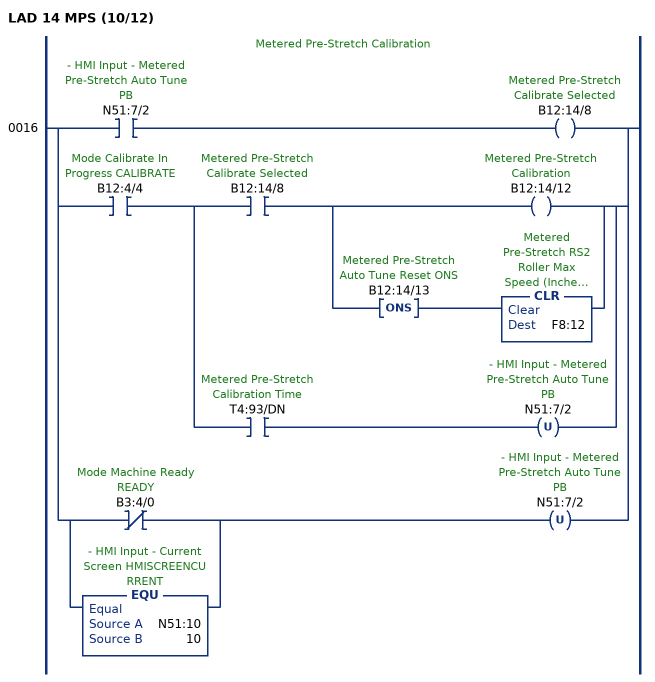
% Rung: 16 %
% Metered Pre-Stretch Calibration %
SOR BST XIC N51:7/2 OTE B12:14/8 NXB XIC B12:4/4 BST XIC B12:14/8 BST OTE B12:14/12 NXB ONS B12:14/13 CLR F8:12 BND NXB XIC T4:93/DN OTU N51:7/2 BND NXB BST XIO B3:4/0 NXB EQU N51:10 10 BND OTU N51:7/2 BND EOR
%   N51:7/2  "- HMI Input - Metered Pre-Stretch Auto Tune PB" %
%   B12:14/8  "Metered Pre-Stretch Calibrate Selected" %
%   B12:4/4  CALIBRATE  "Mode Calibrate In Progress" %
%   B12:14/12  "Metered Pre-Stretch Calibration" %
%   B12:14/13  "Metered Pre-Stretch Auto Tune Reset ONS" %
%   F8:12  RS2MAXSPEED  "Metered Pre-Stretch RS2 Roller Max Speed (Inches Per Second)" %
%   T4:93  "Metered Pre-Stretch Calibration Time" %
%   B3:4/0  READY  "Mode Machine Ready" %
%   N51:10  HMISCREENCURRENT  "- HMI Input - Current Screen" %

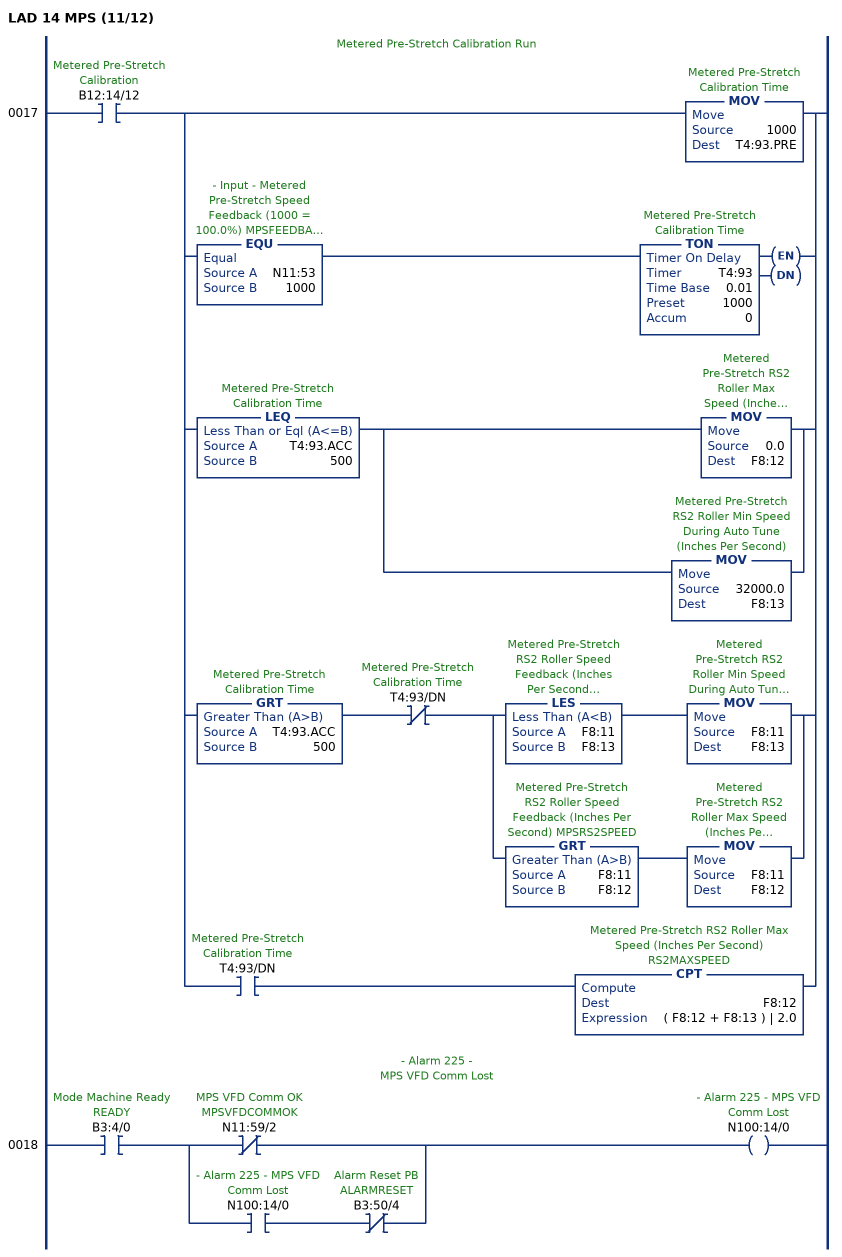
% Rung: 17 %
% Metered Pre-Stretch Calibration Run %
SOR XIC B12:14/12 BST MOV 1000 T4:93.PRE NXB EQU N11:53 1000 TON T4:93 0.01 1000 0 NXB LEQ T4:93.ACC 500 BST MOV 0.0 F8:12 NXB MOV 32000.0 F8:13 BND NXB GRT T4:93.ACC 500 XIO T4:93/DN BST LES F8:11 F8:13 MOV F8:11 F8:13 NXB GRT F8:11 F8:12 MOV F8:11 F8:12 BND NXB XIC T4:93/DN CPT F8:12 " ( F8:12 + F8:13 ) | 2.0 " BND EOR
%   B12:14/12  "Metered Pre-Stretch Calibration" %
%   T4:93  "Metered Pre-Stretch Calibration Time" %
%   N11:53  MPSFEEDBACK  "- Input - Metered Pre-Stretch Speed Feedback (1000 = 100.0%)" %
%   F8:12  RS2MAXSPEED  "Metered Pre-Stretch RS2 Roller Max Speed (Inches Per Second)" %
%   F8:13  "Metered Pre-Stretch RS2 Roller Min Speed During Auto Tune (Inches Per Second)" %
%   F8:11  MPSRS2SPEED  "Metered Pre-Stretch RS2 Roller Speed Feedback (Inches Per Second)" %
% Rung: 18 %
% - Alarm 225 -
% 
% MPS VFD Comm Lost %
SOR XIC B3:4/0 BST XIO N11:59/2 NXB XIC N100:14/0 XIO B3:50/4 BND OTE N100:14/0 EOR
%   B3:4/0  READY  "Mode Machine Ready" %
%   N11:59/2  MPSVFDCOMMOK  "MPS VFD Comm OK" %
%   N100:14/0  "- Alarm 225 - MPS VFD Comm Lost" %
%   B3:50/4  ALARMRESET  "Alarm Reset PB" %

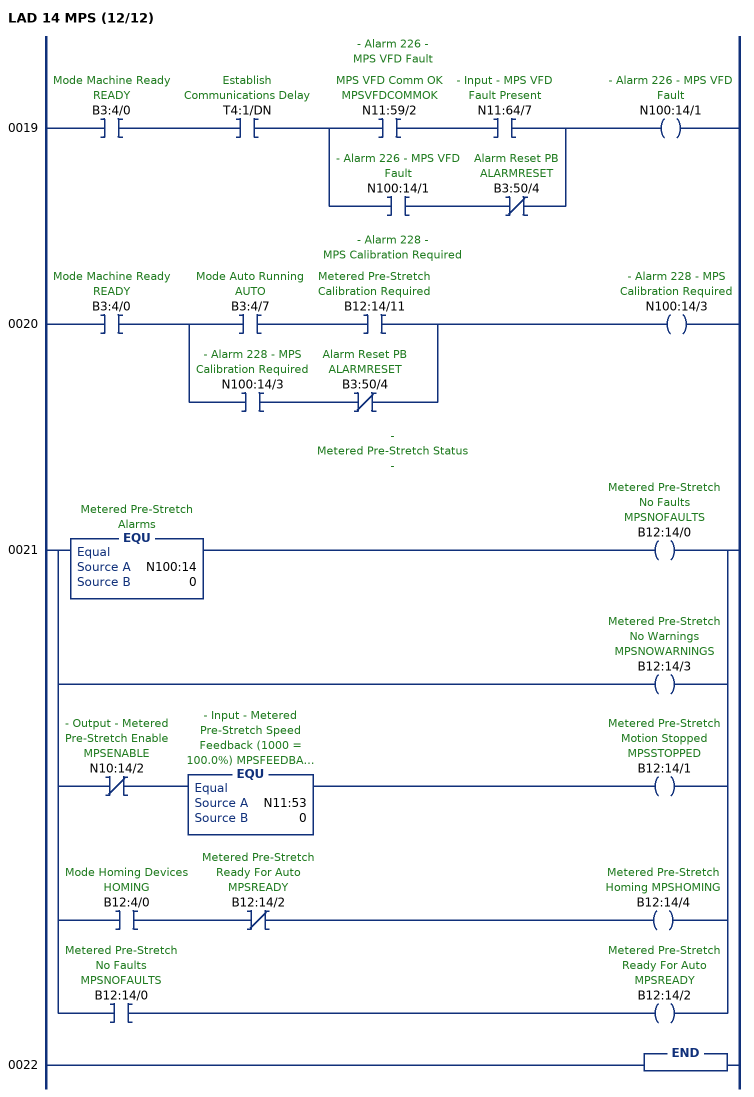
% Rung: 19 %
% - Alarm 226 -
% 
% MPS VFD Fault %
SOR XIC B3:4/0 XIC T4:1/DN BST XIC N11:59/2 XIC N11:64/7 NXB XIC N100:14/1 XIO B3:50/4 BND OTE N100:14/1 EOR
%   B3:4/0  READY  "Mode Machine Ready" %
%   T4:1  "Establish Communications Delay" %
%   N11:59/2  MPSVFDCOMMOK  "MPS VFD Comm OK" %
%   N11:64/7  "- Input - MPS VFD Fault Present" %
%   N100:14/1  "- Alarm 226 - MPS VFD Fault" %
%   B3:50/4  ALARMRESET  "Alarm Reset PB" %
% Rung: 20 %
% - Alarm 228 -
% 
% MPS Calibration Required %
SOR XIC B3:4/0 BST XIC B3:4/7 XIC B12:14/11 NXB XIC N100:14/3 XIO B3:50/4 BND OTE N100:14/3 EOR
%   B3:4/0  READY  "Mode Machine Ready" %
%   B3:4/7  AUTO  "Mode Auto Running" %
%   B12:14/11  "Metered Pre-Stretch Calibration Required" %
%   N100:14/3  "- Alarm 228 - MPS Calibration Required" %
%   B3:50/4  ALARMRESET  "Alarm Reset PB" %
% Rung: 21 %
% -
% 
% Metered Pre-Stretch Status
% 
% - %
SOR BST EQU N100:14 0 OTE B12:14/0 NXB OTE B12:14/3 NXB XIO N10:14/2 EQU N11:53 0 OTE B12:14/1 NXB XIC B12:4/0 XIO B12:14/2 OTE B12:14/4 NXB XIC B12:14/0 OTE B12:14/2 BND EOR
%   N100:14  "Metered Pre-Stretch Alarms" %
%   B12:14/0  MPSNOFAULTS  "Metered Pre-Stretch No Faults" %
%   B12:14/3  MPSNOWARNINGS  "Metered Pre-Stretch No Warnings" %
%   N10:14/2  MPSENABLE  "- Output - Metered Pre-Stretch Enable" %
%   N11:53  MPSFEEDBACK  "- Input - Metered Pre-Stretch Speed Feedback (1000 = 100.0%)" %
%   B12:14/1  MPSSTOPPED  "Metered Pre-Stretch Motion Stopped" %
%   B12:4/0  HOMING  "Mode Homing Devices" %
%   B12:14/2  MPSREADY  "Metered Pre-Stretch Ready For Auto" %
%   B12:14/4  MPSHOMING  "Metered Pre-Stretch Homing" %
% Rung: 22 %
SOR END EOR

LADDER 15 "CUTTER ASM"
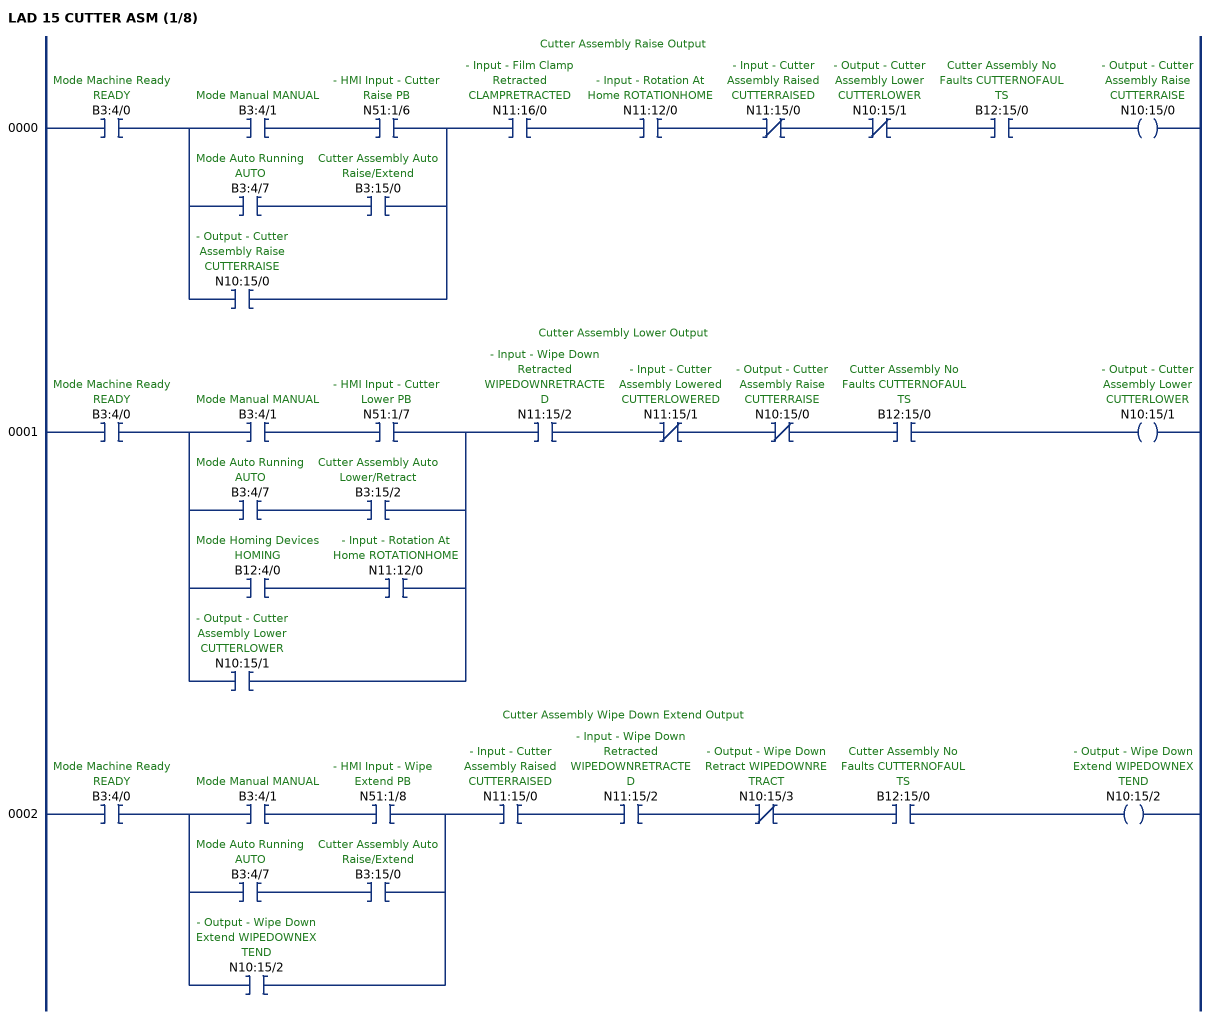
% Rung: 0 %
% Cutter Assembly Raise Output %
SOR XIC B3:4/0 BST XIC B3:4/1 XIC N51:1/6 NXB XIC B3:4/7 XIC B3:15/0 NXB XIC N10:15/0 BND XIC N11:16/0 XIC N11:12/0 XIO N11:15/0 XIO N10:15/1 XIC B12:15/0 OTE N10:15/0 EOR
%   B3:4/0  READY  "Mode Machine Ready" %
%   B3:4/1  MANUAL  "Mode Manual" %
%   N51:1/6  "- HMI Input - Cutter Raise PB" %
%   B3:4/7  AUTO  "Mode Auto Running" %
%   B3:15/0  "Cutter Assembly Auto Raise/Extend" %
%   N10:15/0  CUTTERRAISE  "- Output - Cutter Assembly Raise" %
%   N11:16/0  CLAMPRETRACTED  "- Input - Film Clamp Retracted" %
%   N11:12/0  ROTATIONHOME  "- Input - Rotation At Home" %
%   N11:15/0  CUTTERRAISED  "- Input - Cutter Assembly Raised" %
%   N10:15/1  CUTTERLOWER  "- Output - Cutter Assembly Lower" %
%   B12:15/0  CUTTERNOFAULTS  "Cutter Assembly No Faults" %
% Rung: 1 %
% Cutter Assembly Lower Output %
SOR XIC B3:4/0 BST XIC B3:4/1 XIC N51:1/7 NXB XIC B3:4/7 XIC B3:15/2 NXB XIC B12:4/0 XIC N11:12/0 NXB XIC N10:15/1 BND XIC N11:15/2 XIO N11:15/1 XIO N10:15/0 XIC B12:15/0 OTE N10:15/1 EOR
%   B3:4/0  READY  "Mode Machine Ready" %
%   B3:4/1  MANUAL  "Mode Manual" %
%   N51:1/7  "- HMI Input - Cutter Lower PB" %
%   B3:4/7  AUTO  "Mode Auto Running" %
%   B3:15/2  "Cutter Assembly Auto Lower/Retract" %
%   B12:4/0  HOMING  "Mode Homing Devices" %
%   N11:12/0  ROTATIONHOME  "- Input - Rotation At Home" %
%   N10:15/1  CUTTERLOWER  "- Output - Cutter Assembly Lower" %
%   N11:15/2  WIPEDOWNRETRACTED  "- Input - Wipe Down Retracted" %
%   N11:15/1  CUTTERLOWERED  "- Input - Cutter Assembly Lowered" %
%   N10:15/0  CUTTERRAISE  "- Output - Cutter Assembly Raise" %
%   B12:15/0  CUTTERNOFAULTS  "Cutter Assembly No Faults" %
% Rung: 2 %
% Cutter Assembly Wipe Down Extend Output %
SOR XIC B3:4/0 BST XIC B3:4/1 XIC N51:1/8 NXB XIC B3:4/7 XIC B3:15/0 NXB XIC N10:15/2 BND XIC N11:15/0 XIC N11:15/2 XIO N10:15/3 XIC B12:15/0 OTE N10:15/2 EOR
%   B3:4/0  READY  "Mode Machine Ready" %
%   B3:4/1  MANUAL  "Mode Manual" %
%   N51:1/8  "- HMI Input - Wipe Extend PB" %
%   B3:4/7  AUTO  "Mode Auto Running" %
%   B3:15/0  "Cutter Assembly Auto Raise/Extend" %
%   N10:15/2  WIPEDOWNEXTEND  "- Output - Wipe Down Extend" %
%   N11:15/0  CUTTERRAISED  "- Input - Cutter Assembly Raised" %
%   N11:15/2  WIPEDOWNRETRACTED  "- Input - Wipe Down Retracted" %
%   N10:15/3  WIPEDOWNRETRACT  "- Output - Wipe Down Retract" %
%   B12:15/0  CUTTERNOFAULTS  "Cutter Assembly No Faults" %

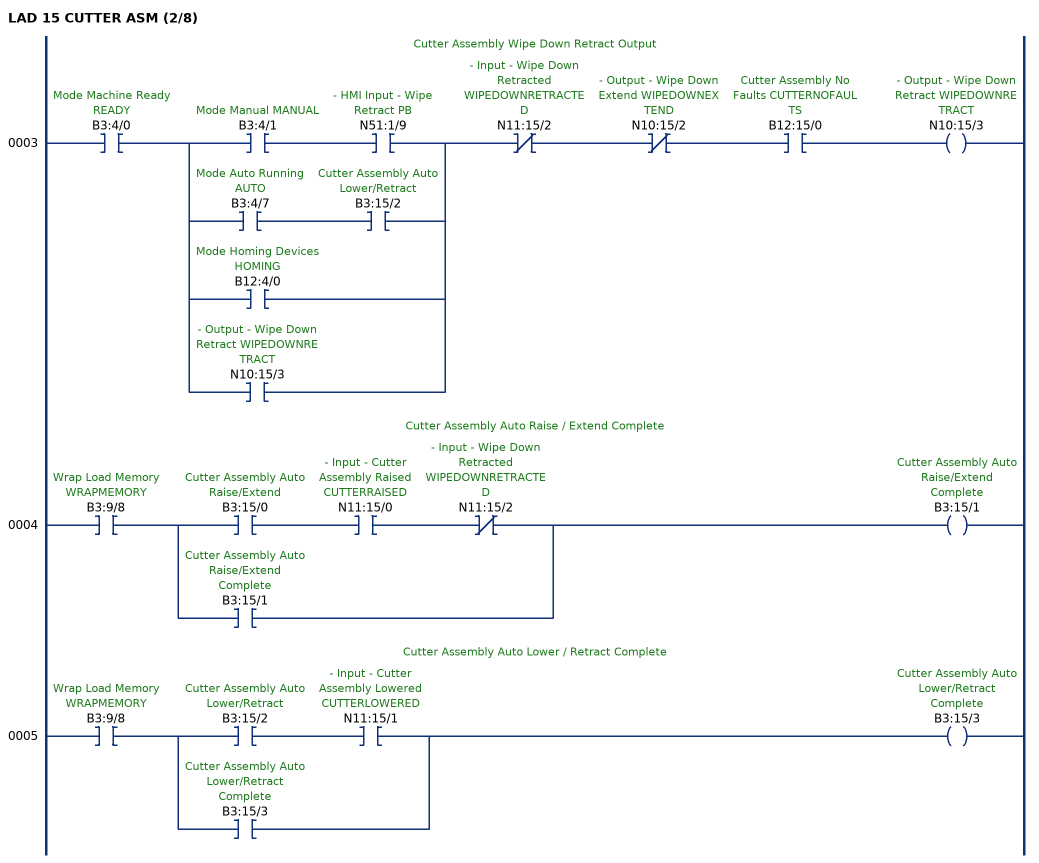
% Rung: 3 %
% Cutter Assembly Wipe Down Retract Output %
SOR XIC B3:4/0 BST XIC B3:4/1 XIC N51:1/9 NXB XIC B3:4/7 XIC B3:15/2 NXB XIC B12:4/0 NXB XIC N10:15/3 BND XIO N11:15/2 XIO N10:15/2 XIC B12:15/0 OTE N10:15/3 EOR
%   B3:4/0  READY  "Mode Machine Ready" %
%   B3:4/1  MANUAL  "Mode Manual" %
%   N51:1/9  "- HMI Input - Wipe Retract PB" %
%   B3:4/7  AUTO  "Mode Auto Running" %
%   B3:15/2  "Cutter Assembly Auto Lower/Retract" %
%   B12:4/0  HOMING  "Mode Homing Devices" %
%   N10:15/3  WIPEDOWNRETRACT  "- Output - Wipe Down Retract" %
%   N11:15/2  WIPEDOWNRETRACTED  "- Input - Wipe Down Retracted" %
%   N10:15/2  WIPEDOWNEXTEND  "- Output - Wipe Down Extend" %
%   B12:15/0  CUTTERNOFAULTS  "Cutter Assembly No Faults" %
% Rung: 4 %
% Cutter Assembly Auto Raise / Extend Complete %
SOR XIC B3:9/8 BST XIC B3:15/0 XIC N11:15/0 XIO N11:15/2 NXB XIC B3:15/1 BND OTE B3:15/1 EOR
%   B3:9/8  WRAPMEMORY  "Wrap Load Memory" %
%   B3:15/0  "Cutter Assembly Auto Raise/Extend" %
%   N11:15/0  CUTTERRAISED  "- Input - Cutter Assembly Raised" %
%   N11:15/2  WIPEDOWNRETRACTED  "- Input - Wipe Down Retracted" %
%   B3:15/1  "Cutter Assembly Auto Raise/Extend Complete" %
% Rung: 5 %
% Cutter Assembly Auto Lower / Retract Complete %
SOR XIC B3:9/8 BST XIC B3:15/2 XIC N11:15/1 NXB XIC B3:15/3 BND OTE B3:15/3 EOR
%   B3:9/8  WRAPMEMORY  "Wrap Load Memory" %
%   B3:15/2  "Cutter Assembly Auto Lower/Retract" %
%   N11:15/1  CUTTERLOWERED  "- Input - Cutter Assembly Lowered" %
%   B3:15/3  "Cutter Assembly Auto Lower/Retract Complete" %

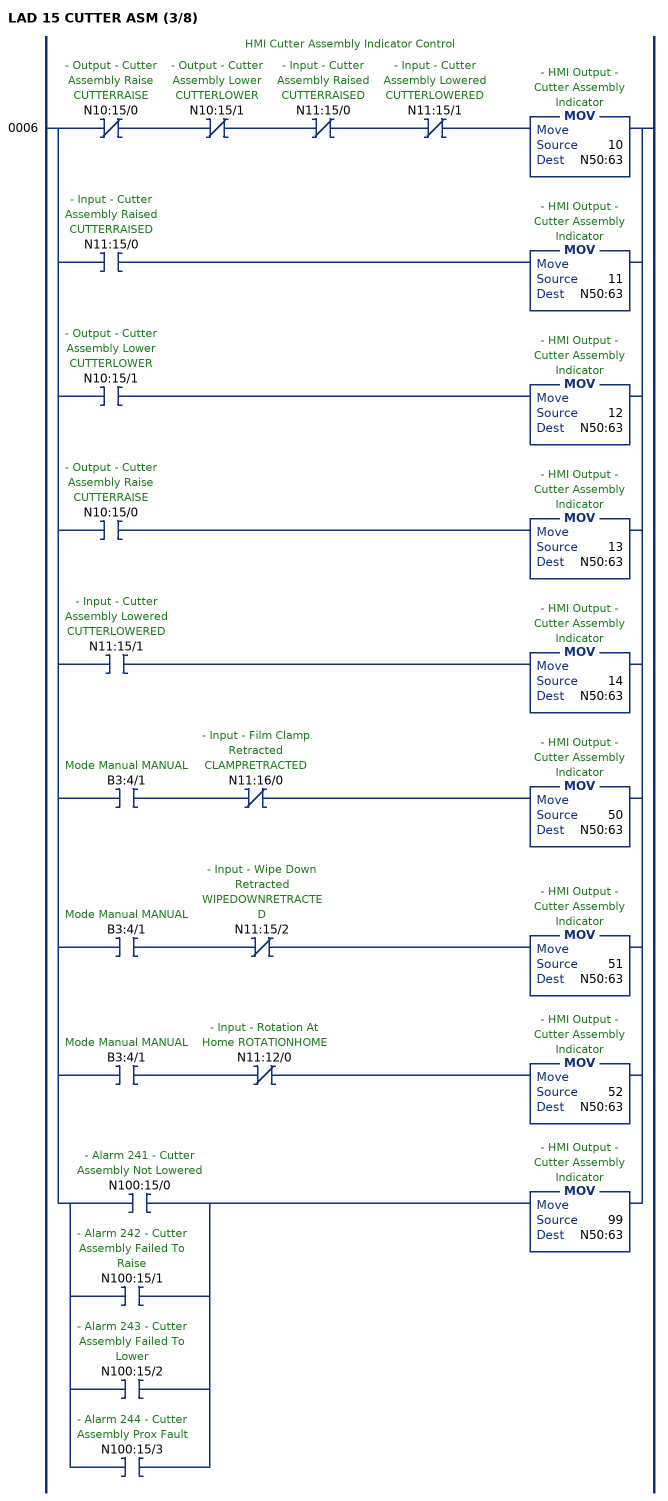
% Rung: 6 %
% HMI Cutter Assembly Indicator Control %
SOR BST XIO N10:15/0 XIO N10:15/1 XIO N11:15/0 XIO N11:15/1 MOV 10 N50:63 NXB XIC N11:15/0 MOV 11 N50:63 NXB XIC N10:15/1 MOV 12 N50:63 NXB XIC N10:15/0 MOV 13 N50:63 NXB XIC N11:15/1 MOV 14 N50:63 NXB XIC B3:4/1 XIO N11:16/0 MOV 50 N50:63 NXB XIC B3:4/1 XIO N11:15/2 MOV 51 N50:63 NXB XIC B3:4/1 XIO N11:12/0 MOV 52 N50:63 NXB BST XIC N100:15/0 NXB XIC N100:15/1 NXB XIC N100:15/2 NXB XIC N100:15/3 BND MOV 99 N50:63 BND EOR
%   N10:15/0  CUTTERRAISE  "- Output - Cutter Assembly Raise" %
%   N10:15/1  CUTTERLOWER  "- Output - Cutter Assembly Lower" %
%   N11:15/0  CUTTERRAISED  "- Input - Cutter Assembly Raised" %
%   N11:15/1  CUTTERLOWERED  "- Input - Cutter Assembly Lowered" %
%   N50:63  "- HMI Output - Cutter Assembly Indicator" %
%   B3:4/1  MANUAL  "Mode Manual" %
%   N11:16/0  CLAMPRETRACTED  "- Input - Film Clamp Retracted" %
%   N11:15/2  WIPEDOWNRETRACTED  "- Input - Wipe Down Retracted" %
%   N11:12/0  ROTATIONHOME  "- Input - Rotation At Home" %
%   N100:15/0  "- Alarm 241 - Cutter Assembly Not Lowered" %
%   N100:15/1  "- Alarm 242 - Cutter Assembly Failed To Raise" %
%   N100:15/2  "- Alarm 243 - Cutter Assembly Failed To Lower" %
%   N100:15/3  "- Alarm 244 - Cutter Assembly Prox Fault" %

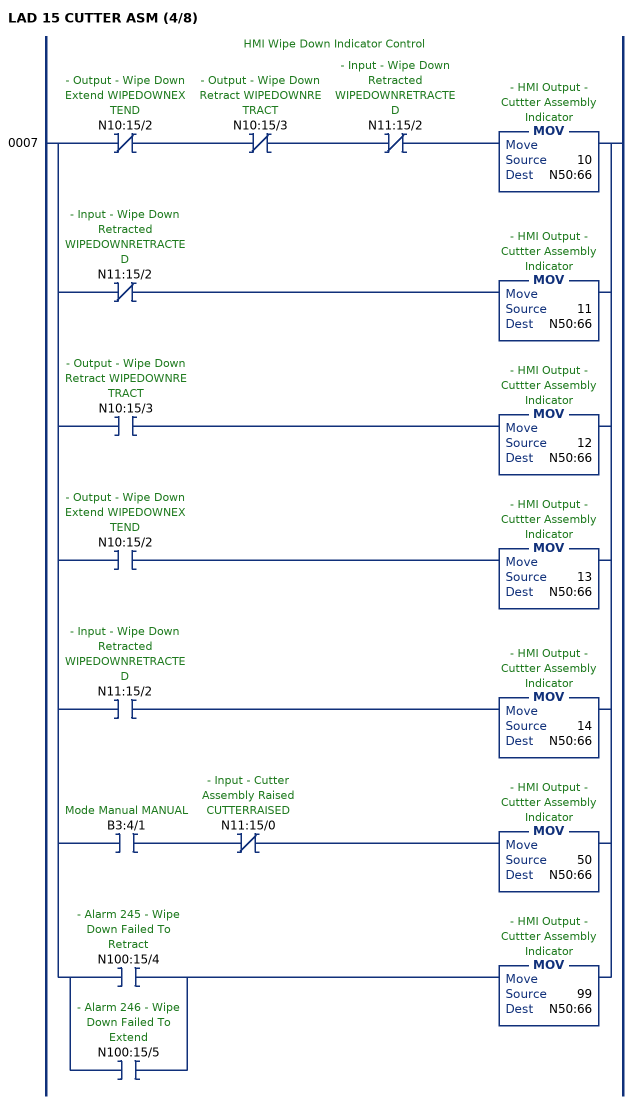
% Rung: 7 %
% HMI Wipe Down Indicator Control %
SOR BST XIO N10:15/2 XIO N10:15/3 XIO N11:15/2 MOV 10 N50:66 NXB XIO N11:15/2 MOV 11 N50:66 NXB XIC N10:15/3 MOV 12 N50:66 NXB XIC N10:15/2 MOV 13 N50:66 NXB XIC N11:15/2 MOV 14 N50:66 NXB XIC B3:4/1 XIO N11:15/0 MOV 50 N50:66 NXB BST XIC N100:15/4 NXB XIC N100:15/5 BND MOV 99 N50:66 BND EOR
%   N10:15/2  WIPEDOWNEXTEND  "- Output - Wipe Down Extend" %
%   N10:15/3  WIPEDOWNRETRACT  "- Output - Wipe Down Retract" %
%   N11:15/2  WIPEDOWNRETRACTED  "- Input - Wipe Down Retracted" %
%   N50:66  "- HMI Output - Cuttter Assembly Indicator" %
%   B3:4/1  MANUAL  "Mode Manual" %
%   N11:15/0  CUTTERRAISED  "- Input - Cutter Assembly Raised" %
%   N100:15/4  "- Alarm 245 - Wipe Down Failed To Retract" %
%   N100:15/5  "- Alarm 246 - Wipe Down Failed To Extend" %

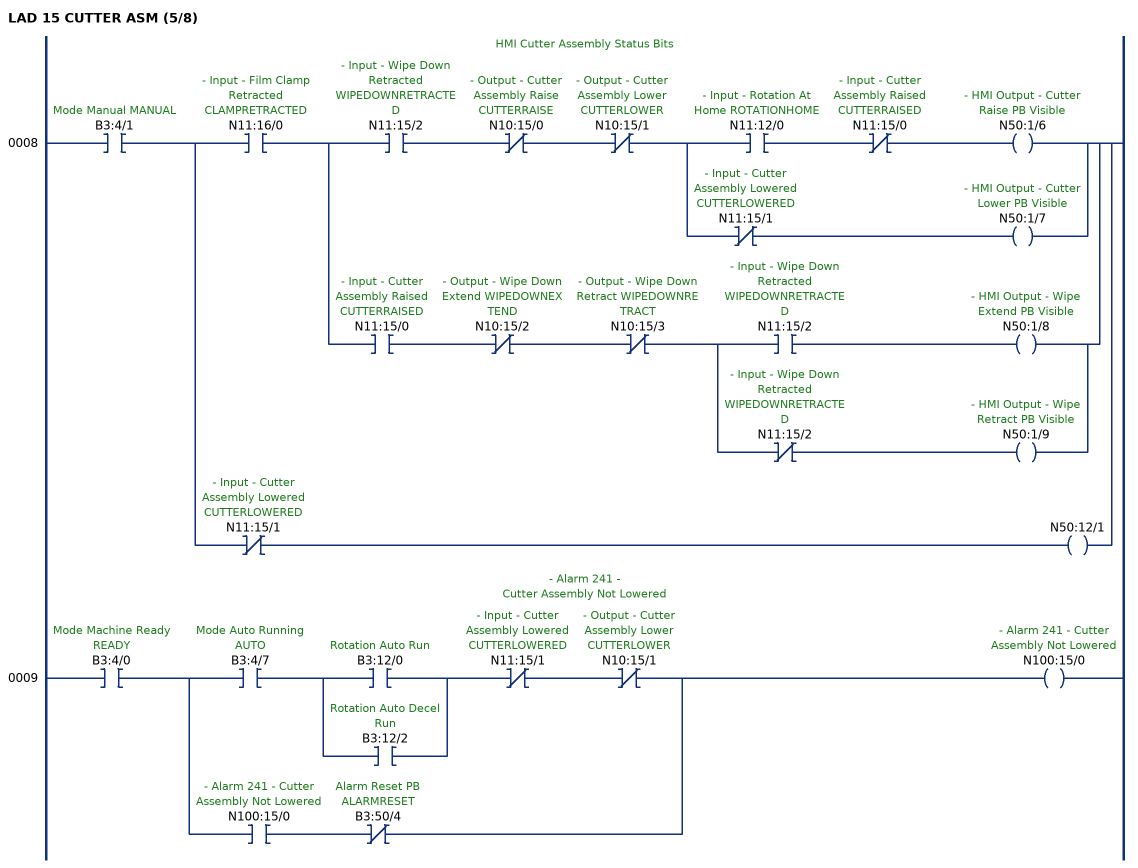
% Rung: 8 %
% HMI Cutter Assembly Status Bits %
SOR XIC B3:4/1 BST XIC N11:16/0 BST XIC N11:15/2 XIO N10:15/0 XIO N10:15/1 BST XIC N11:12/0 XIO N11:15/0 OTE N50:1/6 NXB XIO N11:15/1 OTE N50:1/7 BND NXB XIC N11:15/0 XIO N10:15/2 XIO N10:15/3 BST XIC N11:15/2 OTE N50:1/8 NXB XIO N11:15/2 OTE N50:1/9 BND BND NXB XIO N11:15/1 OTE N50:12/1 BND EOR
%   B3:4/1  MANUAL  "Mode Manual" %
%   N11:16/0  CLAMPRETRACTED  "- Input - Film Clamp Retracted" %
%   N11:15/2  WIPEDOWNRETRACTED  "- Input - Wipe Down Retracted" %
%   N10:15/0  CUTTERRAISE  "- Output - Cutter Assembly Raise" %
%   N10:15/1  CUTTERLOWER  "- Output - Cutter Assembly Lower" %
%   N11:12/0  ROTATIONHOME  "- Input - Rotation At Home" %
%   N11:15/0  CUTTERRAISED  "- Input - Cutter Assembly Raised" %
%   N50:1/6  "- HMI Output - Cutter Raise PB Visible" %
%   N11:15/1  CUTTERLOWERED  "- Input - Cutter Assembly Lowered" %
%   N50:1/7  "- HMI Output - Cutter Lower PB Visible" %
%   N10:15/2  WIPEDOWNEXTEND  "- Output - Wipe Down Extend" %
%   N10:15/3  WIPEDOWNRETRACT  "- Output - Wipe Down Retract" %
%   N50:1/8  "- HMI Output - Wipe Extend PB Visible" %
%   N50:1/9  "- HMI Output - Wipe Retract PB Visible" %
% Rung: 9 %
% - Alarm 241 -
% 
% Cutter Assembly Not Lowered %
SOR XIC B3:4/0 BST XIC B3:4/7 BST XIC B3:12/0 NXB XIC B3:12/2 BND XIO N11:15/1 XIO N10:15/1 NXB XIC N100:15/0 XIO B3:50/4 BND OTE N100:15/0 EOR
%   B3:4/0  READY  "Mode Machine Ready" %
%   B3:4/7  AUTO  "Mode Auto Running" %
%   B3:12/0  "Rotation Auto Run" %
%   B3:12/2  "Rotation Auto Decel Run" %
%   N11:15/1  CUTTERLOWERED  "- Input - Cutter Assembly Lowered" %
%   N10:15/1  CUTTERLOWER  "- Output - Cutter Assembly Lower" %
%   N100:15/0  "- Alarm 241 - Cutter Assembly Not Lowered" %
%   B3:50/4  ALARMRESET  "Alarm Reset PB" %

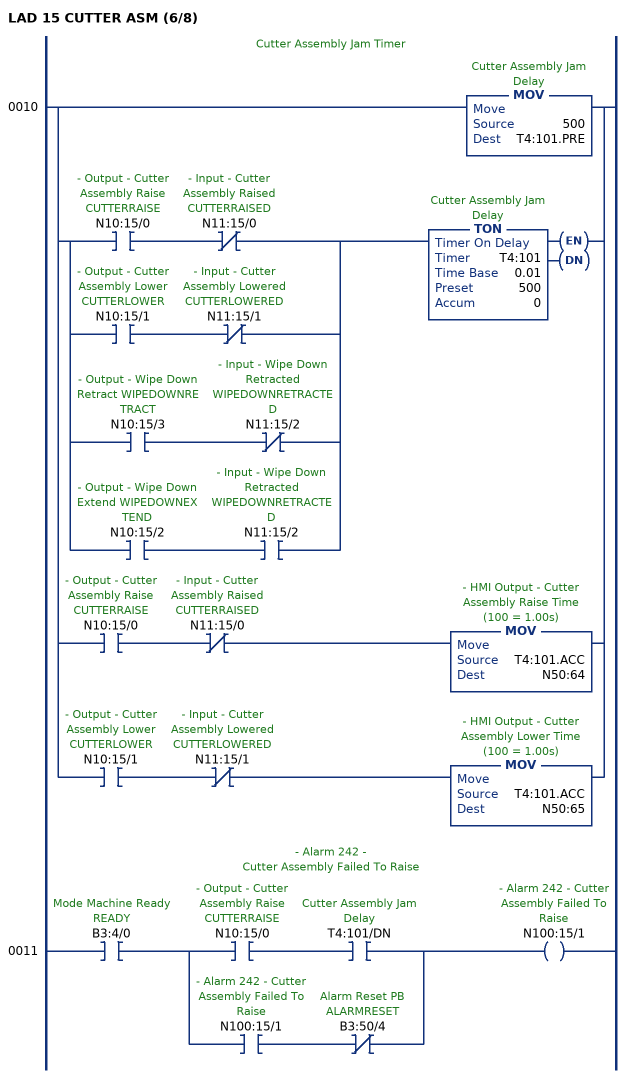
% Rung: 10 %
% Cutter Assembly Jam Timer %
SOR BST MOV 500 T4:101.PRE NXB BST XIC N10:15/0 XIO N11:15/0 NXB XIC N10:15/1 XIO N11:15/1 NXB XIC N10:15/3 XIO N11:15/2 NXB XIC N10:15/2 XIC N11:15/2 BND TON T4:101 0.01 500 0 NXB XIC N10:15/0 XIO N11:15/0 MOV T4:101.ACC N50:64 NXB XIC N10:15/1 XIO N11:15/1 MOV T4:101.ACC N50:65 BND EOR
%   T4:101  "Cutter Assembly Jam Delay" %
%   N10:15/0  CUTTERRAISE  "- Output - Cutter Assembly Raise" %
%   N11:15/0  CUTTERRAISED  "- Input - Cutter Assembly Raised" %
%   N10:15/1  CUTTERLOWER  "- Output - Cutter Assembly Lower" %
%   N11:15/1  CUTTERLOWERED  "- Input - Cutter Assembly Lowered" %
%   N10:15/3  WIPEDOWNRETRACT  "- Output - Wipe Down Retract" %
%   N11:15/2  WIPEDOWNRETRACTED  "- Input - Wipe Down Retracted" %
%   N10:15/2  WIPEDOWNEXTEND  "- Output - Wipe Down Extend" %
%   N50:64  "- HMI Output - Cutter Assembly Raise Time (100 = 1.00s)" %
%   N50:65  "- HMI Output - Cutter Assembly Lower Time (100 = 1.00s)" %
% Rung: 11 %
% - Alarm 242 -
% 
% Cutter Assembly Failed To Raise %
SOR XIC B3:4/0 BST XIC N10:15/0 XIC T4:101/DN NXB XIC N100:15/1 XIO B3:50/4 BND OTE N100:15/1 EOR
%   B3:4/0  READY  "Mode Machine Ready" %
%   N10:15/0  CUTTERRAISE  "- Output - Cutter Assembly Raise" %
%   T4:101  "Cutter Assembly Jam Delay" %
%   N100:15/1  "- Alarm 242 - Cutter Assembly Failed To Raise" %
%   B3:50/4  ALARMRESET  "Alarm Reset PB" %

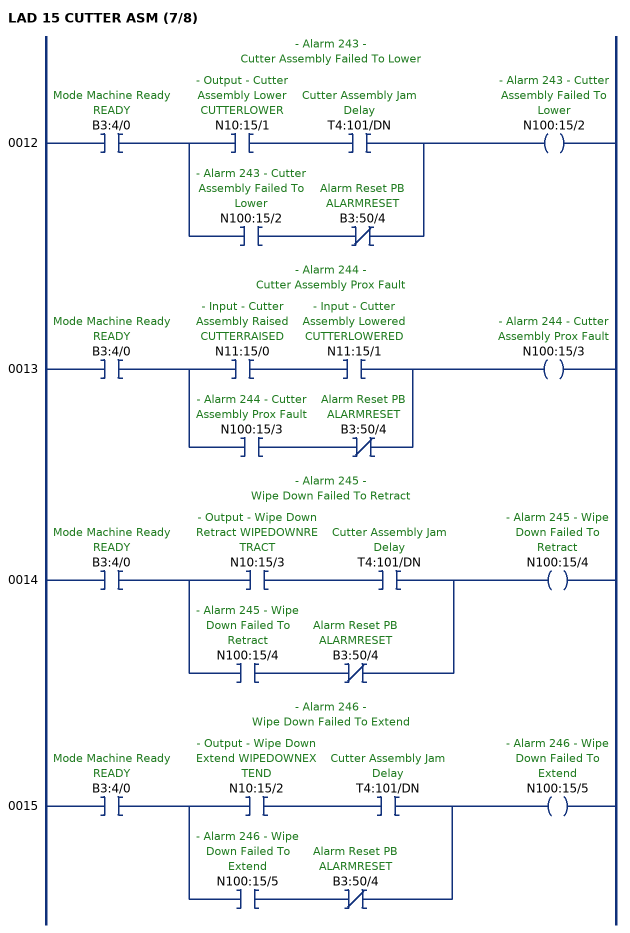
% Rung: 12 %
% - Alarm 243 -
% 
% Cutter Assembly Failed To Lower %
SOR XIC B3:4/0 BST XIC N10:15/1 XIC T4:101/DN NXB XIC N100:15/2 XIO B3:50/4 BND OTE N100:15/2 EOR
%   B3:4/0  READY  "Mode Machine Ready" %
%   N10:15/1  CUTTERLOWER  "- Output - Cutter Assembly Lower" %
%   T4:101  "Cutter Assembly Jam Delay" %
%   N100:15/2  "- Alarm 243 - Cutter Assembly Failed To Lower" %
%   B3:50/4  ALARMRESET  "Alarm Reset PB" %
% Rung: 13 %
% - Alarm 244 -
% 
% Cutter Assembly Prox Fault %
SOR XIC B3:4/0 BST XIC N11:15/0 XIC N11:15/1 NXB XIC N100:15/3 XIO B3:50/4 BND OTE N100:15/3 EOR
%   B3:4/0  READY  "Mode Machine Ready" %
%   N11:15/0  CUTTERRAISED  "- Input - Cutter Assembly Raised" %
%   N11:15/1  CUTTERLOWERED  "- Input - Cutter Assembly Lowered" %
%   N100:15/3  "- Alarm 244 - Cutter Assembly Prox Fault" %
%   B3:50/4  ALARMRESET  "Alarm Reset PB" %
% Rung: 14 %
% - Alarm 245 -
% 
% Wipe Down Failed To Retract %
SOR XIC B3:4/0 BST XIC N10:15/3 XIC T4:101/DN NXB XIC N100:15/4 XIO B3:50/4 BND OTE N100:15/4 EOR
%   B3:4/0  READY  "Mode Machine Ready" %
%   N10:15/3  WIPEDOWNRETRACT  "- Output - Wipe Down Retract" %
%   T4:101  "Cutter Assembly Jam Delay" %
%   N100:15/4  "- Alarm 245 - Wipe Down Failed To Retract" %
%   B3:50/4  ALARMRESET  "Alarm Reset PB" %
% Rung: 15 %
% - Alarm 246 -
% 
% Wipe Down Failed To Extend %
SOR XIC B3:4/0 BST XIC N10:15/2 XIC T4:101/DN NXB XIC N100:15/5 XIO B3:50/4 BND OTE N100:15/5 EOR
%   B3:4/0  READY  "Mode Machine Ready" %
%   N10:15/2  WIPEDOWNEXTEND  "- Output - Wipe Down Extend" %
%   T4:101  "Cutter Assembly Jam Delay" %
%   N100:15/5  "- Alarm 246 - Wipe Down Failed To Extend" %
%   B3:50/4  ALARMRESET  "Alarm Reset PB" %

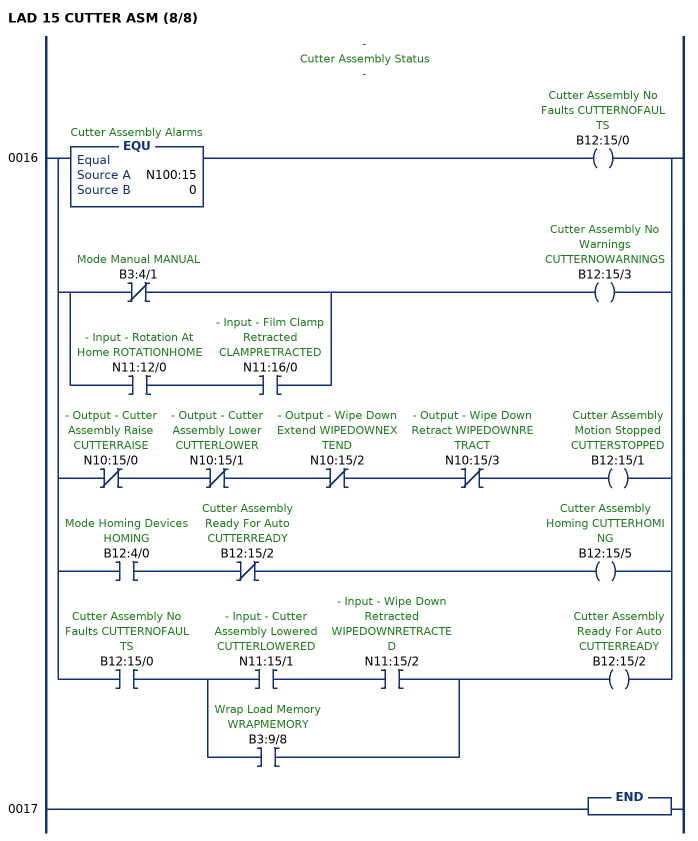
% Rung: 16 %
% -
% 
% Cutter Assembly Status
% 
% - %
SOR BST EQU N100:15 0 OTE B12:15/0 NXB BST XIO B3:4/1 NXB XIC N11:12/0 XIC N11:16/0 BND OTE B12:15/3 NXB XIO N10:15/0 XIO N10:15/1 XIO N10:15/2 XIO N10:15/3 OTE B12:15/1 NXB XIC B12:4/0 XIO B12:15/2 OTE B12:15/5 NXB XIC B12:15/0 BST XIC N11:15/1 XIC N11:15/2 NXB XIC B3:9/8 BND OTE B12:15/2 BND EOR
%   N100:15  "Cutter Assembly Alarms" %
%   B12:15/0  CUTTERNOFAULTS  "Cutter Assembly No Faults" %
%   B3:4/1  MANUAL  "Mode Manual" %
%   N11:12/0  ROTATIONHOME  "- Input - Rotation At Home" %
%   N11:16/0  CLAMPRETRACTED  "- Input - Film Clamp Retracted" %
%   B12:15/3  CUTTERNOWARNINGS  "Cutter Assembly No Warnings" %
%   N10:15/0  CUTTERRAISE  "- Output - Cutter Assembly Raise" %
%   N10:15/1  CUTTERLOWER  "- Output - Cutter Assembly Lower" %
%   N10:15/2  WIPEDOWNEXTEND  "- Output - Wipe Down Extend" %
%   N10:15/3  WIPEDOWNRETRACT  "- Output - Wipe Down Retract" %
%   B12:15/1  CUTTERSTOPPED  "Cutter Assembly Motion Stopped" %
%   B12:4/0  HOMING  "Mode Homing Devices" %
%   B12:15/2  CUTTERREADY  "Cutter Assembly Ready For Auto" %
%   B12:15/5  CUTTERHOMING  "Cutter Assembly Homing" %
%   N11:15/1  CUTTERLOWERED  "- Input - Cutter Assembly Lowered" %
%   N11:15/2  WIPEDOWNRETRACTED  "- Input - Wipe Down Retracted" %
%   B3:9/8  WRAPMEMORY  "Wrap Load Memory" %
% Rung: 17 %
SOR END EOR

LADDER 16 "FILM CLAMP"
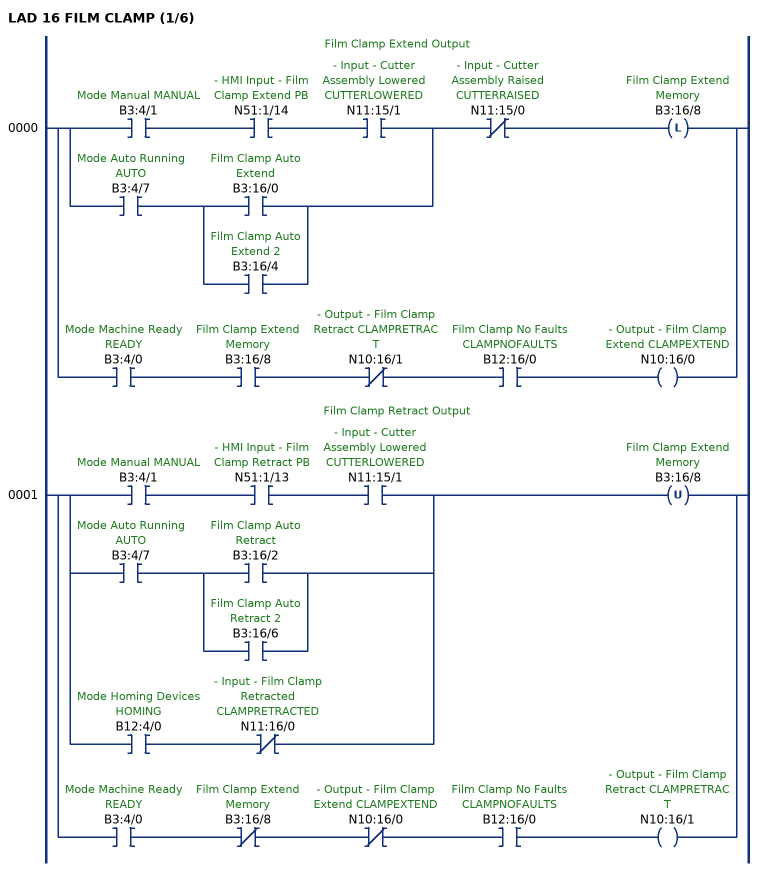
% Rung: 0 %
% Film Clamp Extend Output %
SOR BST BST XIC B3:4/1 XIC N51:1/14 XIC N11:15/1 NXB XIC B3:4/7 BST XIC B3:16/0 NXB XIC B3:16/4 BND BND XIO N11:15/0 OTL B3:16/8 NXB XIC B3:4/0 XIC B3:16/8 XIO N10:16/1 XIC B12:16/0 OTE N10:16/0 BND EOR
%   B3:4/1  MANUAL  "Mode Manual" %
%   N51:1/14  "- HMI Input - Film Clamp Extend PB" %
%   N11:15/1  CUTTERLOWERED  "- Input - Cutter Assembly Lowered" %
%   B3:4/7  AUTO  "Mode Auto Running" %
%   B3:16/0  "Film Clamp Auto Extend" %
%   B3:16/4  "Film Clamp Auto Extend 2" %
%   N11:15/0  CUTTERRAISED  "- Input - Cutter Assembly Raised" %
%   B3:16/8  "Film Clamp Extend Memory" %
%   B3:4/0  READY  "Mode Machine Ready" %
%   N10:16/1  CLAMPRETRACT  "- Output - Film Clamp Retract" %
%   B12:16/0  CLAMPNOFAULTS  "Film Clamp No Faults" %
%   N10:16/0  CLAMPEXTEND  "- Output - Film Clamp Extend" %
% Rung: 1 %
% Film Clamp Retract Output %
SOR BST BST XIC B3:4/1 XIC N51:1/13 XIC N11:15/1 NXB XIC B3:4/7 BST XIC B3:16/2 NXB XIC B3:16/6 BND NXB XIC B12:4/0 XIO N11:16/0 BND OTU B3:16/8 NXB XIC B3:4/0 XIO B3:16/8 XIO N10:16/0 XIC B12:16/0 OTE N10:16/1 BND EOR
%   B3:4/1  MANUAL  "Mode Manual" %
%   N51:1/13  "- HMI Input - Film Clamp Retract PB" %
%   N11:15/1  CUTTERLOWERED  "- Input - Cutter Assembly Lowered" %
%   B3:4/7  AUTO  "Mode Auto Running" %
%   B3:16/2  "Film Clamp Auto Retract" %
%   B3:16/6  "Film Clamp Auto Retract 2" %
%   B12:4/0  HOMING  "Mode Homing Devices" %
%   N11:16/0  CLAMPRETRACTED  "- Input - Film Clamp Retracted" %
%   B3:16/8  "Film Clamp Extend Memory" %
%   B3:4/0  READY  "Mode Machine Ready" %
%   N10:16/0  CLAMPEXTEND  "- Output - Film Clamp Extend" %
%   B12:16/0  CLAMPNOFAULTS  "Film Clamp No Faults" %
%   N10:16/1  CLAMPRETRACT  "- Output - Film Clamp Retract" %

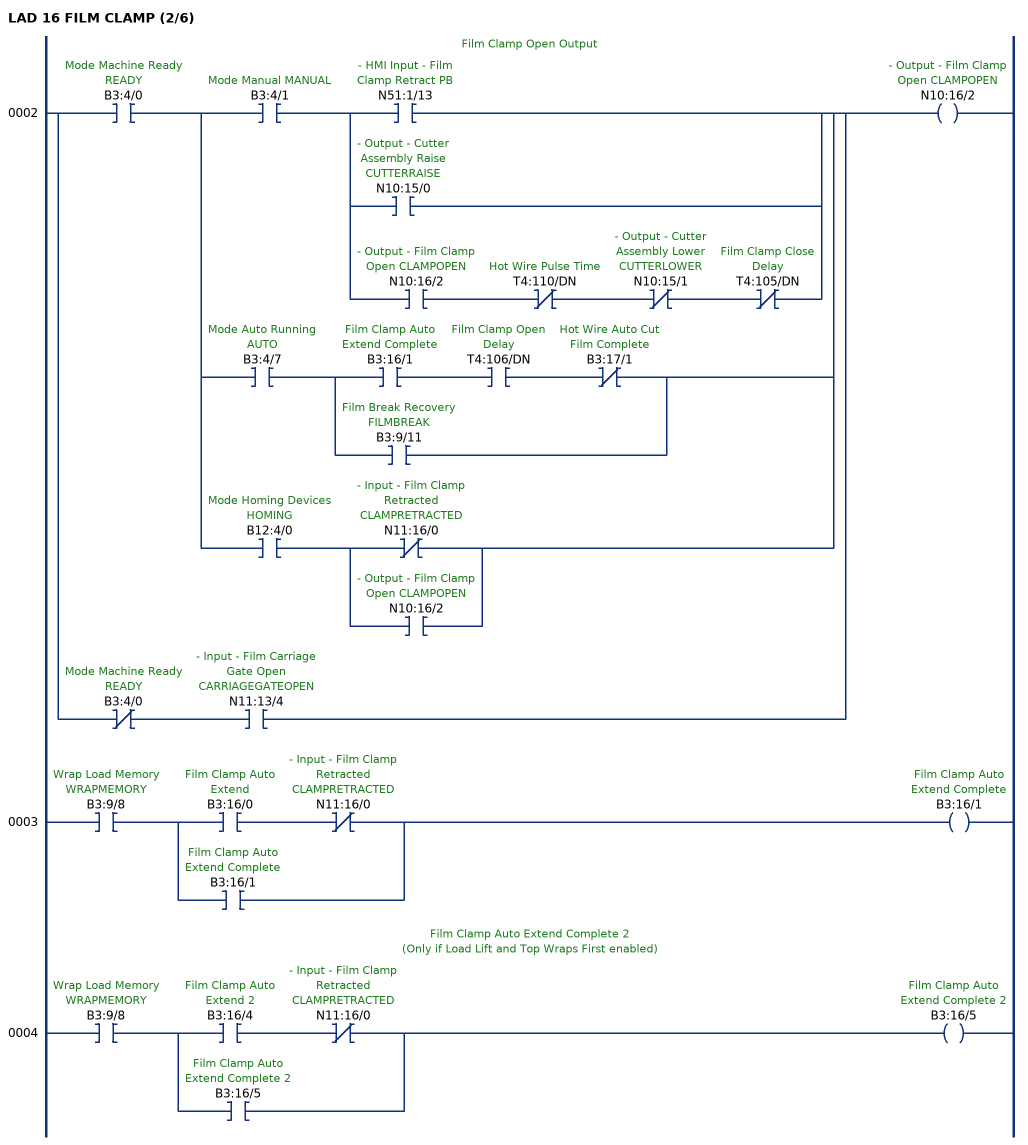
% Rung: 2 %
% Film Clamp Open Output %
SOR BST XIC B3:4/0 BST XIC B3:4/1 BST XIC N51:1/13 NXB XIC N10:15/0 NXB XIC N10:16/2 XIO T4:110/DN XIO N10:15/1 XIO T4:105/DN BND NXB XIC B3:4/7 BST XIC B3:16/1 XIC T4:106/DN XIO B3:17/1 NXB XIC B3:9/11 BND NXB XIC B12:4/0 BST XIO N11:16/0 NXB XIC N10:16/2 BND BND NXB XIO B3:4/0 XIC N11:13/4 BND OTE N10:16/2 EOR
%   B3:4/0  READY  "Mode Machine Ready" %
%   B3:4/1  MANUAL  "Mode Manual" %
%   N51:1/13  "- HMI Input - Film Clamp Retract PB" %
%   N10:15/0  CUTTERRAISE  "- Output - Cutter Assembly Raise" %
%   N10:16/2  CLAMPOPEN  "- Output - Film Clamp Open" %
%   T4:110  "Hot Wire Pulse Time" %
%   N10:15/1  CUTTERLOWER  "- Output - Cutter Assembly Lower" %
%   T4:105  "Film Clamp Close Delay" %
%   B3:4/7  AUTO  "Mode Auto Running" %
%   B3:16/1  "Film Clamp Auto Extend Complete" %
%   T4:106  "Film Clamp Open Delay" %
%   B3:17/1  "Hot Wire Auto Cut Film Complete" %
%   B3:9/11  FILMBREAK  "Film Break Recovery" %
%   B12:4/0  HOMING  "Mode Homing Devices" %
%   N11:16/0  CLAMPRETRACTED  "- Input - Film Clamp Retracted" %
%   N11:13/4  CARRIAGEGATEOPEN  "- Input - Film Carriage Gate Open" %
% Rung: 3 %
SOR XIC B3:9/8 BST XIC B3:16/0 XIO N11:16/0 NXB XIC B3:16/1 BND OTE B3:16/1 EOR
%   B3:9/8  WRAPMEMORY  "Wrap Load Memory" %
%   B3:16/0  "Film Clamp Auto Extend" %
%   N11:16/0  CLAMPRETRACTED  "- Input - Film Clamp Retracted" %
%   B3:16/1  "Film Clamp Auto Extend Complete" %
% Rung: 4 %
% Film Clamp Auto Extend Complete 2
% (Only if Load Lift and Top Wraps First enabled) %
SOR XIC B3:9/8 BST XIC B3:16/4 XIO N11:16/0 NXB XIC B3:16/5 BND OTE B3:16/5 EOR
%   B3:9/8  WRAPMEMORY  "Wrap Load Memory" %
%   B3:16/4  "Film Clamp Auto Extend 2" %
%   N11:16/0  CLAMPRETRACTED  "- Input - Film Clamp Retracted" %
%   B3:16/5  "Film Clamp Auto Extend Complete 2" %

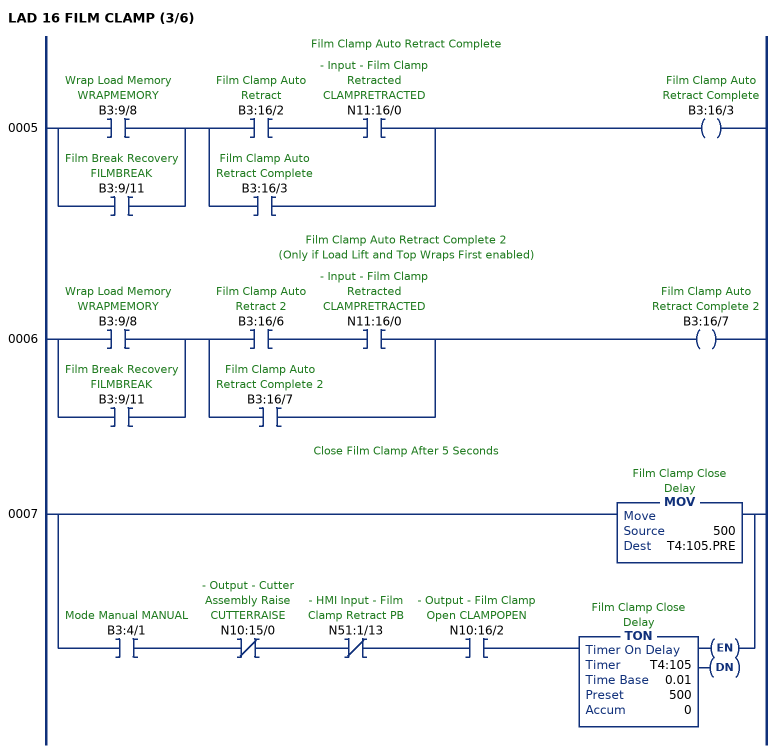
% Rung: 5 %
% Film Clamp Auto Retract Complete %
SOR BST XIC B3:9/8 NXB XIC B3:9/11 BND BST XIC B3:16/2 XIC N11:16/0 NXB XIC B3:16/3 BND OTE B3:16/3 EOR
%   B3:9/8  WRAPMEMORY  "Wrap Load Memory" %
%   B3:9/11  FILMBREAK  "Film Break Recovery" %
%   B3:16/2  "Film Clamp Auto Retract" %
%   N11:16/0  CLAMPRETRACTED  "- Input - Film Clamp Retracted" %
%   B3:16/3  "Film Clamp Auto Retract Complete" %
% Rung: 6 %
% Film Clamp Auto Retract Complete 2
% (Only if Load Lift and Top Wraps First enabled) %
SOR BST XIC B3:9/8 NXB XIC B3:9/11 BND BST XIC B3:16/6 XIC N11:16/0 NXB XIC B3:16/7 BND OTE B3:16/7 EOR
%   B3:9/8  WRAPMEMORY  "Wrap Load Memory" %
%   B3:9/11  FILMBREAK  "Film Break Recovery" %
%   B3:16/6  "Film Clamp Auto Retract 2" %
%   N11:16/0  CLAMPRETRACTED  "- Input - Film Clamp Retracted" %
%   B3:16/7  "Film Clamp Auto Retract Complete 2" %
% Rung: 7 %
% Close Film Clamp After 5 Seconds %
SOR BST MOV 500 T4:105.PRE NXB XIC B3:4/1 XIO N10:15/0 XIO N51:1/13 XIC N10:16/2 TON T4:105 0.01 500 0 BND EOR
%   T4:105  "Film Clamp Close Delay" %
%   B3:4/1  MANUAL  "Mode Manual" %
%   N10:15/0  CUTTERRAISE  "- Output - Cutter Assembly Raise" %
%   N51:1/13  "- HMI Input - Film Clamp Retract PB" %
%   N10:16/2  CLAMPOPEN  "- Output - Film Clamp Open" %

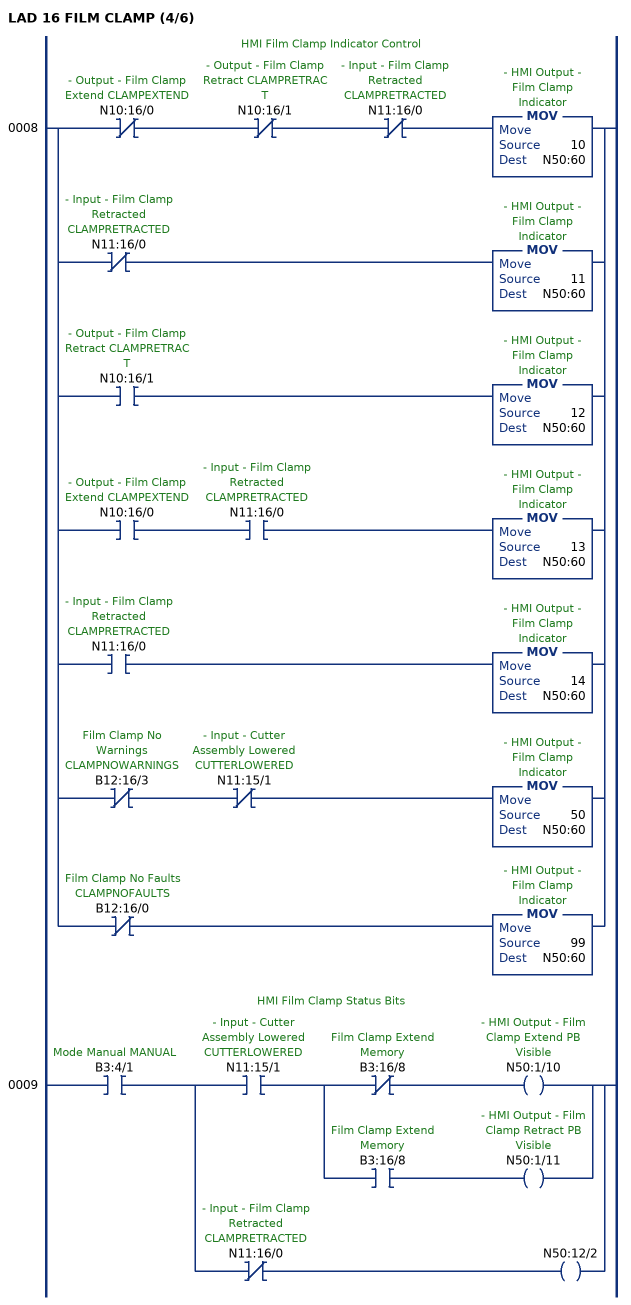
% Rung: 8 %
% HMI Film Clamp Indicator Control %
SOR BST XIO N10:16/0 XIO N10:16/1 XIO N11:16/0 MOV 10 N50:60 NXB XIO N11:16/0 MOV 11 N50:60 NXB XIC N10:16/1 MOV 12 N50:60 NXB XIC N10:16/0 XIC N11:16/0 MOV 13 N50:60 NXB XIC N11:16/0 MOV 14 N50:60 NXB XIO B12:16/3 XIO N11:15/1 MOV 50 N50:60 NXB XIO B12:16/0 MOV 99 N50:60 BND EOR
%   N10:16/0  CLAMPEXTEND  "- Output - Film Clamp Extend" %
%   N10:16/1  CLAMPRETRACT  "- Output - Film Clamp Retract" %
%   N11:16/0  CLAMPRETRACTED  "- Input - Film Clamp Retracted" %
%   N50:60  "- HMI Output - Film Clamp Indicator" %
%   B12:16/3  CLAMPNOWARNINGS  "Film Clamp No Warnings" %
%   N11:15/1  CUTTERLOWERED  "- Input - Cutter Assembly Lowered" %
%   B12:16/0  CLAMPNOFAULTS  "Film Clamp No Faults" %
% Rung: 9 %
% HMI Film Clamp Status Bits %
SOR XIC B3:4/1 BST XIC N11:15/1 BST XIO B3:16/8 OTE N50:1/10 NXB XIC B3:16/8 OTE N50:1/11 BND NXB XIO N11:16/0 OTE N50:12/2 BND EOR
%   B3:4/1  MANUAL  "Mode Manual" %
%   N11:15/1  CUTTERLOWERED  "- Input - Cutter Assembly Lowered" %
%   B3:16/8  "Film Clamp Extend Memory" %
%   N50:1/10  "- HMI Output - Film Clamp Extend PB Visible" %
%   N50:1/11  "- HMI Output - Film Clamp Retract PB Visible" %
%   N11:16/0  CLAMPRETRACTED  "- Input - Film Clamp Retracted" %

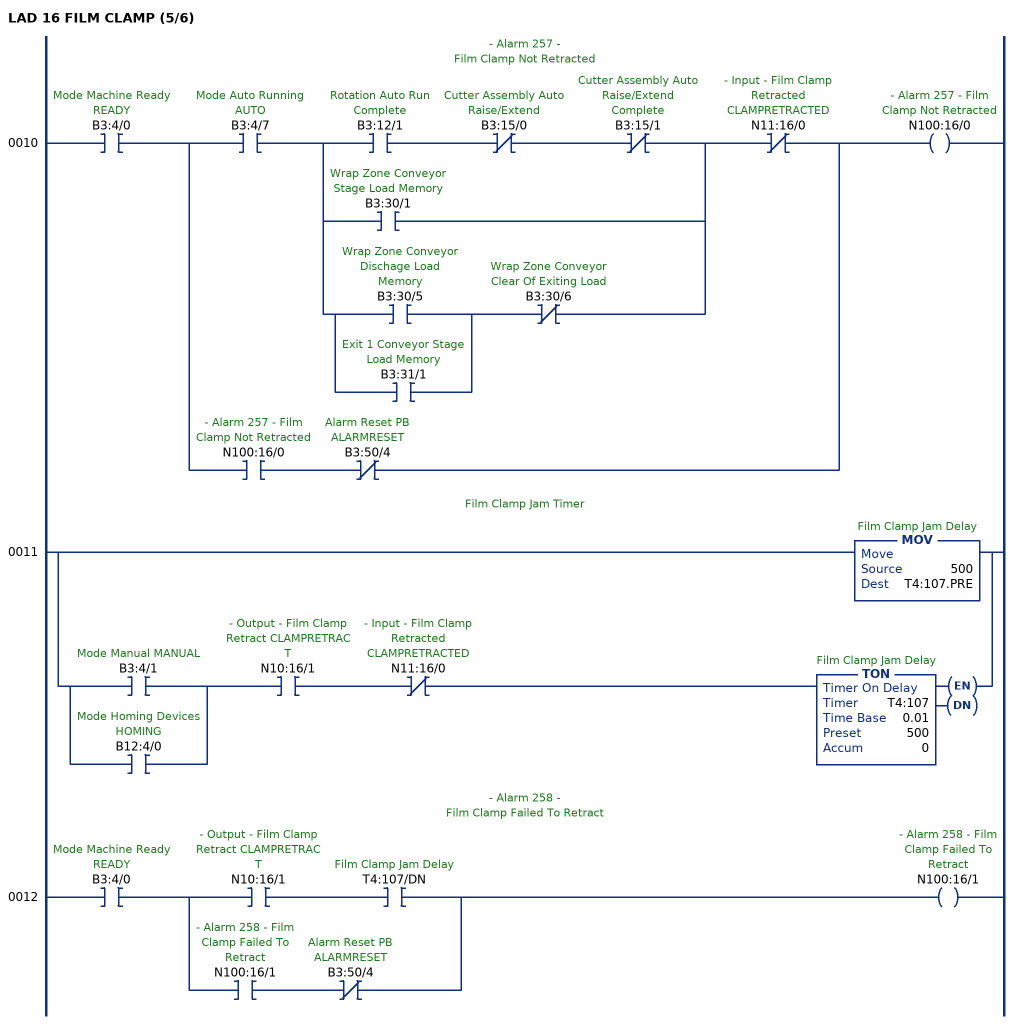
% Rung: 10 %
% - Alarm 257 -
% 
% Film Clamp Not Retracted %
SOR XIC B3:4/0 BST XIC B3:4/7 BST XIC B3:12/1 XIO B3:15/0 XIO B3:15/1 NXB XIC B3:30/1 NXB BST XIC B3:30/5 NXB XIC B3:31/1 BND XIO B3:30/6 BND XIO N11:16/0 NXB XIC N100:16/0 XIO B3:50/4 BND OTE N100:16/0 EOR
%   B3:4/0  READY  "Mode Machine Ready" %
%   B3:4/7  AUTO  "Mode Auto Running" %
%   B3:12/1  "Rotation Auto Run Complete" %
%   B3:15/0  "Cutter Assembly Auto Raise/Extend" %
%   B3:15/1  "Cutter Assembly Auto Raise/Extend Complete" %
%   B3:30/1  "Wrap Zone Conveyor Stage Load Memory" %
%   B3:30/5  "Wrap Zone Conveyor Dischage Load Memory" %
%   B3:31/1  "Exit 1 Conveyor Stage Load Memory" %
%   B3:30/6  "Wrap Zone Conveyor Clear Of Exiting Load" %
%   N11:16/0  CLAMPRETRACTED  "- Input - Film Clamp Retracted" %
%   N100:16/0  "- Alarm 257 - Film Clamp Not Retracted" %
%   B3:50/4  ALARMRESET  "Alarm Reset PB" %
% Rung: 11 %
% Film Clamp Jam Timer %
SOR BST MOV 500 T4:107.PRE NXB BST XIC B3:4/1 NXB XIC B12:4/0 BND XIC N10:16/1 XIO N11:16/0 TON T4:107 0.01 500 0 BND EOR
%   T4:107  "Film Clamp Jam Delay" %
%   B3:4/1  MANUAL  "Mode Manual" %
%   B12:4/0  HOMING  "Mode Homing Devices" %
%   N10:16/1  CLAMPRETRACT  "- Output - Film Clamp Retract" %
%   N11:16/0  CLAMPRETRACTED  "- Input - Film Clamp Retracted" %
% Rung: 12 %
% - Alarm 258 -
% 
% Film Clamp Failed To Retract %
SOR XIC B3:4/0 BST XIC N10:16/1 XIC T4:107/DN NXB XIC N100:16/1 XIO B3:50/4 BND OTE N100:16/1 EOR
%   B3:4/0  READY  "Mode Machine Ready" %
%   N10:16/1  CLAMPRETRACT  "- Output - Film Clamp Retract" %
%   T4:107  "Film Clamp Jam Delay" %
%   N100:16/1  "- Alarm 258 - Film Clamp Failed To Retract" %
%   B3:50/4  ALARMRESET  "Alarm Reset PB" %

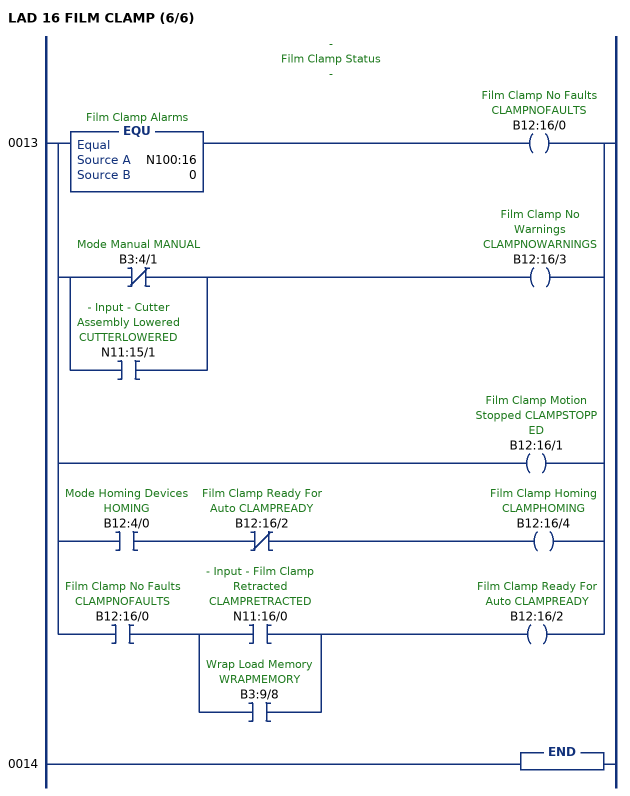
% Rung: 13 %
% -
% 
% Film Clamp Status
% 
% - %
SOR BST EQU N100:16 0 OTE B12:16/0 NXB BST XIO B3:4/1 NXB XIC N11:15/1 BND OTE B12:16/3 NXB OTE B12:16/1 NXB XIC B12:4/0 XIO B12:16/2 OTE B12:16/4 NXB XIC B12:16/0 BST XIC N11:16/0 NXB XIC B3:9/8 BND OTE B12:16/2 BND EOR
%   N100:16  "Film Clamp Alarms" %
%   B12:16/0  CLAMPNOFAULTS  "Film Clamp No Faults" %
%   B3:4/1  MANUAL  "Mode Manual" %
%   N11:15/1  CUTTERLOWERED  "- Input - Cutter Assembly Lowered" %
%   B12:16/3  CLAMPNOWARNINGS  "Film Clamp No Warnings" %
%   B12:16/1  CLAMPSTOPPED  "Film Clamp Motion Stopped" %
%   B12:4/0  HOMING  "Mode Homing Devices" %
%   B12:16/2  CLAMPREADY  "Film Clamp Ready For Auto" %
%   B12:16/4  CLAMPHOMING  "Film Clamp Homing" %
%   N11:16/0  CLAMPRETRACTED  "- Input - Film Clamp Retracted" %
%   B3:9/8  WRAPMEMORY  "Wrap Load Memory" %
% Rung: 14 %
SOR END EOR

LADDER 17 "HOT WIRE"
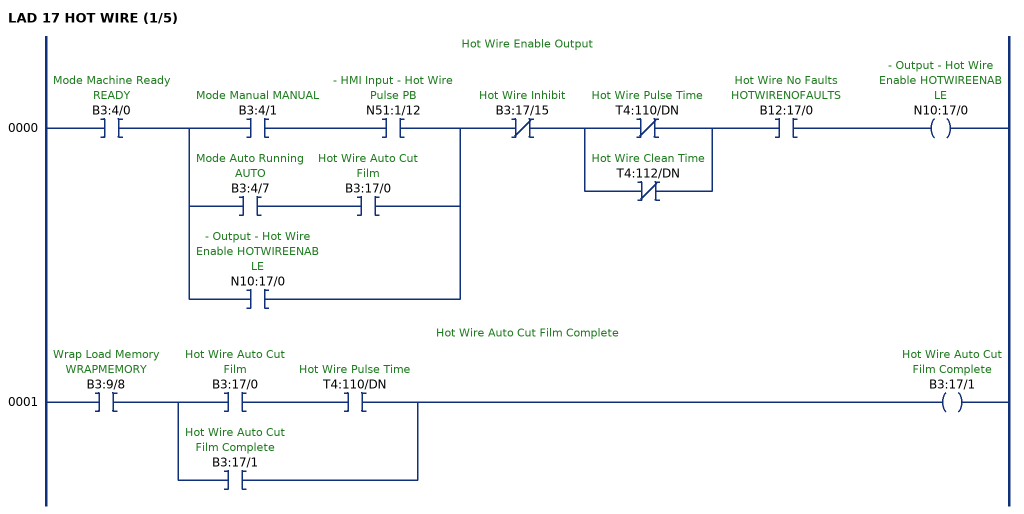
% Rung: 0 %
% Hot Wire Enable Output %
SOR XIC B3:4/0 BST XIC B3:4/1 XIC N51:1/12 NXB XIC B3:4/7 XIC B3:17/0 NXB XIC N10:17/0 BND XIO B3:17/15 BST XIO T4:110/DN NXB XIO T4:112/DN BND XIC B12:17/0 OTE N10:17/0 EOR
%   B3:4/0  READY  "Mode Machine Ready" %
%   B3:4/1  MANUAL  "Mode Manual" %
%   N51:1/12  "- HMI Input - Hot Wire Pulse PB" %
%   B3:4/7  AUTO  "Mode Auto Running" %
%   B3:17/0  "Hot Wire Auto Cut Film" %
%   N10:17/0  HOTWIREENABLE  "- Output - Hot Wire Enable" %
%   B3:17/15  "Hot Wire Inhibit" %
%   T4:110  "Hot Wire Pulse Time" %
%   T4:112  "Hot Wire Clean Time" %
%   B12:17/0  HOTWIRENOFAULTS  "Hot Wire No Faults" %
% Rung: 1 %
% Hot Wire Auto Cut Film Complete %
SOR XIC B3:9/8 BST XIC B3:17/0 XIC T4:110/DN NXB XIC B3:17/1 BND OTE B3:17/1 EOR
%   B3:9/8  WRAPMEMORY  "Wrap Load Memory" %
%   B3:17/0  "Hot Wire Auto Cut Film" %
%   T4:110  "Hot Wire Pulse Time" %
%   B3:17/1  "Hot Wire Auto Cut Film Complete" %

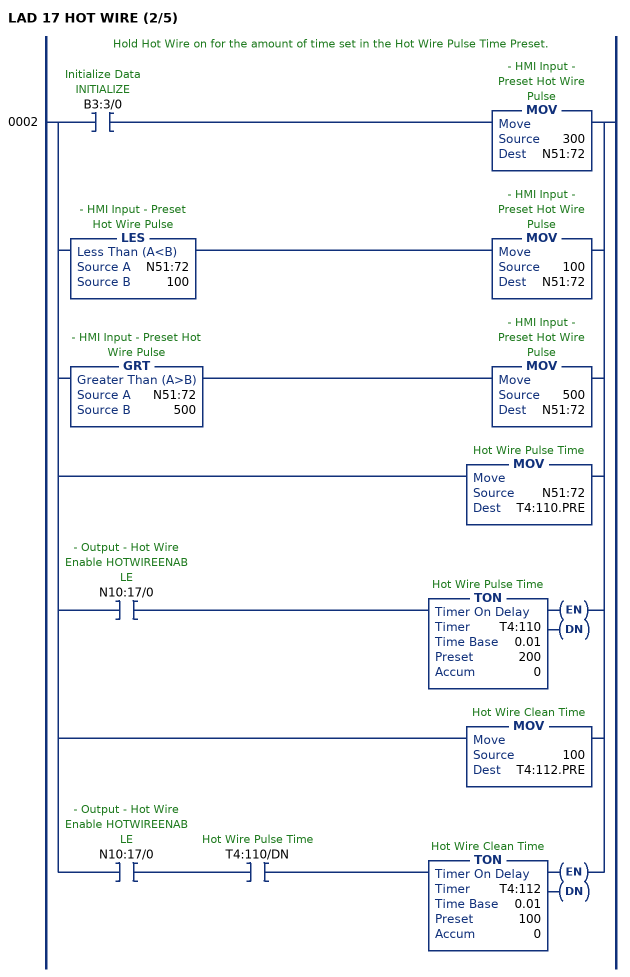
% Rung: 2 %
% Hold Hot Wire on for the amount of time set in the Hot Wire Pulse Time Preset. %
SOR BST BST XIC B3:3/0 MOV 300 N51:72 NXB LES N51:72 100 MOV 100 N51:72 NXB GRT N51:72 500 MOV 500 N51:72 BND NXB MOV N51:72 T4:110.PRE NXB XIC N10:17/0 TON T4:110 0.01 200 0 NXB MOV 100 T4:112.PRE NXB XIC N10:17/0 XIC T4:110/DN TON T4:112 0.01 100 0 BND EOR
%   B3:3/0  INITIALIZE  "Initialize Data" %
%   N51:72  "- HMI Input - Preset Hot Wire Pulse" %
%   T4:110  "Hot Wire Pulse Time" %
%   N10:17/0  HOTWIREENABLE  "- Output - Hot Wire Enable" %
%   T4:112  "Hot Wire Clean Time" %

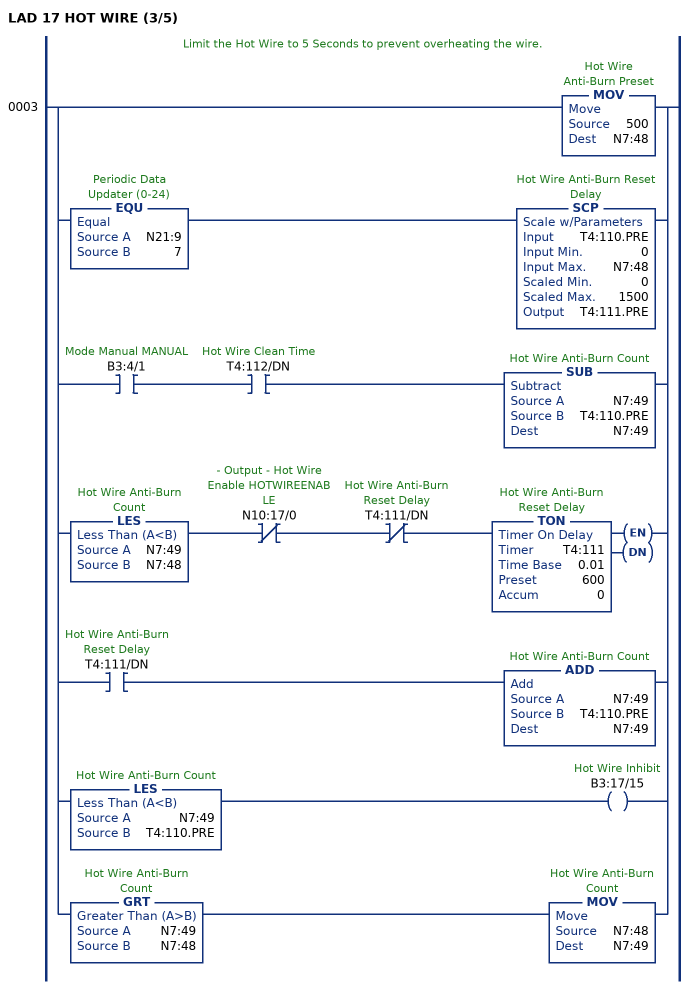
% Rung: 3 %
% Limit the Hot Wire to 5 Seconds to prevent overheating the wire. %
SOR BST MOV 500 N7:48 NXB EQU N21:9 7 SCP T4:110.PRE 0 N7:48 0 1500 T4:111.PRE NXB XIC B3:4/1 XIC T4:112/DN SUB N7:49 T4:110.PRE N7:49 NXB LES N7:49 N7:48 XIO N10:17/0 XIO T4:111/DN TON T4:111 0.01 600 0 NXB XIC T4:111/DN ADD N7:49 T4:110.PRE N7:49 NXB LES N7:49 T4:110.PRE OTE B3:17/15 NXB GRT N7:49 N7:48 MOV N7:48 N7:49 BND EOR
%   N7:48  "Hot Wire Anti-Burn Preset" %
%   N21:9  "Periodic Data Updater (0-24)" %
%   T4:110  "Hot Wire Pulse Time" %
%   T4:111  "Hot Wire Anti-Burn Reset Delay" %
%   B3:4/1  MANUAL  "Mode Manual" %
%   T4:112  "Hot Wire Clean Time" %
%   N7:49  "Hot Wire Anti-Burn Count" %
%   N10:17/0  HOTWIREENABLE  "- Output - Hot Wire Enable" %
%   B3:17/15  "Hot Wire Inhibit" %

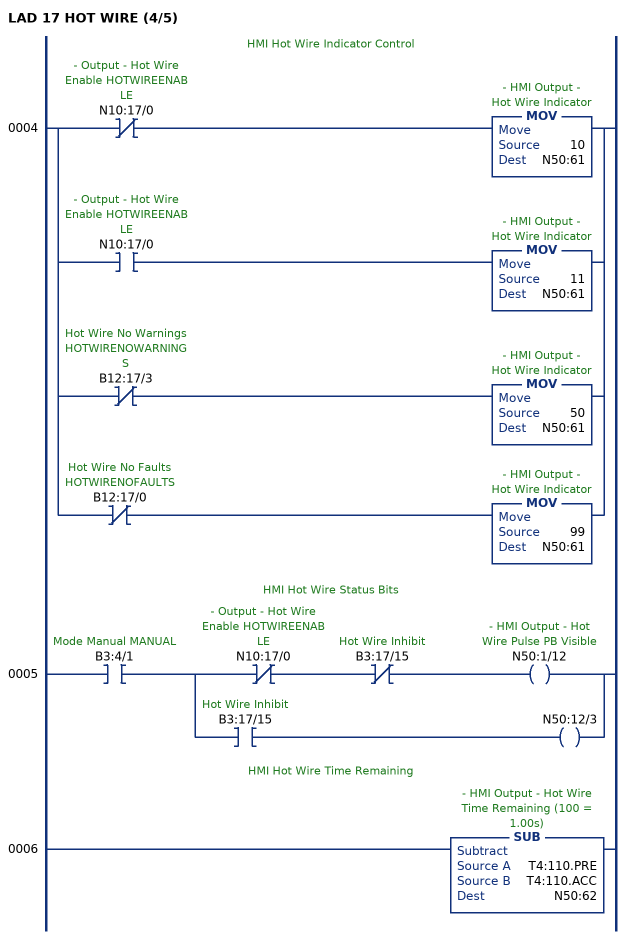
% Rung: 4 %
% HMI Hot Wire Indicator Control %
SOR BST XIO N10:17/0 MOV 10 N50:61 NXB XIC N10:17/0 MOV 11 N50:61 NXB XIO B12:17/3 MOV 50 N50:61 NXB XIO B12:17/0 MOV 99 N50:61 BND EOR
%   N10:17/0  HOTWIREENABLE  "- Output - Hot Wire Enable" %
%   N50:61  "- HMI Output - Hot Wire Indicator" %
%   B12:17/3  HOTWIRENOWARNINGS  "Hot Wire No Warnings" %
%   B12:17/0  HOTWIRENOFAULTS  "Hot Wire No Faults" %
% Rung: 5 %
% HMI Hot Wire Status Bits %
SOR XIC B3:4/1 BST XIO N10:17/0 XIO B3:17/15 OTE N50:1/12 NXB XIC B3:17/15 OTE N50:12/3 BND EOR
%   B3:4/1  MANUAL  "Mode Manual" %
%   N10:17/0  HOTWIREENABLE  "- Output - Hot Wire Enable" %
%   B3:17/15  "Hot Wire Inhibit" %
%   N50:1/12  "- HMI Output - Hot Wire Pulse PB Visible" %
% Rung: 6 %
% HMI Hot Wire Time Remaining %
SOR SUB T4:110.PRE T4:110.ACC N50:62 EOR
%   T4:110  "Hot Wire Pulse Time" %
%   N50:62  "- HMI Output - Hot Wire Time Remaining (100 = 1.00s)" %

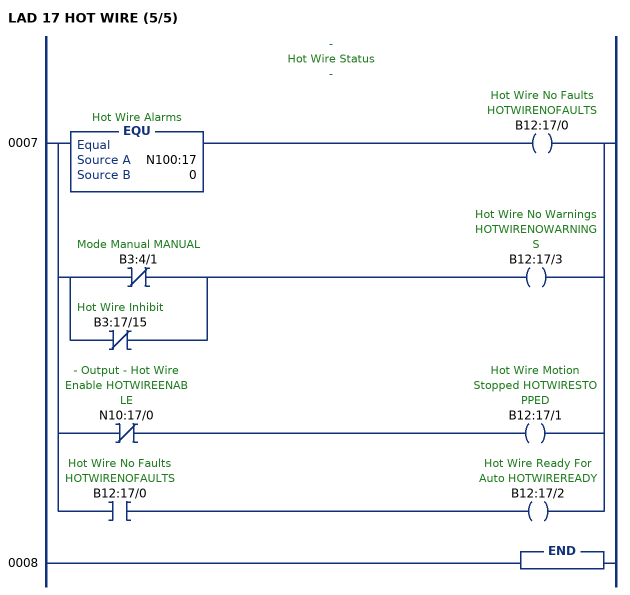
% Rung: 7 %
% -
% 
% Hot Wire Status
% 
% - %
SOR BST EQU N100:17 0 OTE B12:17/0 NXB BST XIO B3:4/1 NXB XIO B3:17/15 BND OTE B12:17/3 NXB XIO N10:17/0 OTE B12:17/1 NXB XIC B12:17/0 OTE B12:17/2 BND EOR
%   N100:17  "Hot Wire Alarms" %
%   B12:17/0  HOTWIRENOFAULTS  "Hot Wire No Faults" %
%   B3:4/1  MANUAL  "Mode Manual" %
%   B3:17/15  "Hot Wire Inhibit" %
%   B12:17/3  HOTWIRENOWARNINGS  "Hot Wire No Warnings" %
%   N10:17/0  HOTWIREENABLE  "- Output - Hot Wire Enable" %
%   B12:17/1  HOTWIRESTOPPED  "Hot Wire Motion Stopped" %
%   B12:17/2  HOTWIREREADY  "Hot Wire Ready For Auto" %
% Rung: 8 %
SOR END EOR

LADDER 19 "TSD"    % Top Sheet Dispenser %
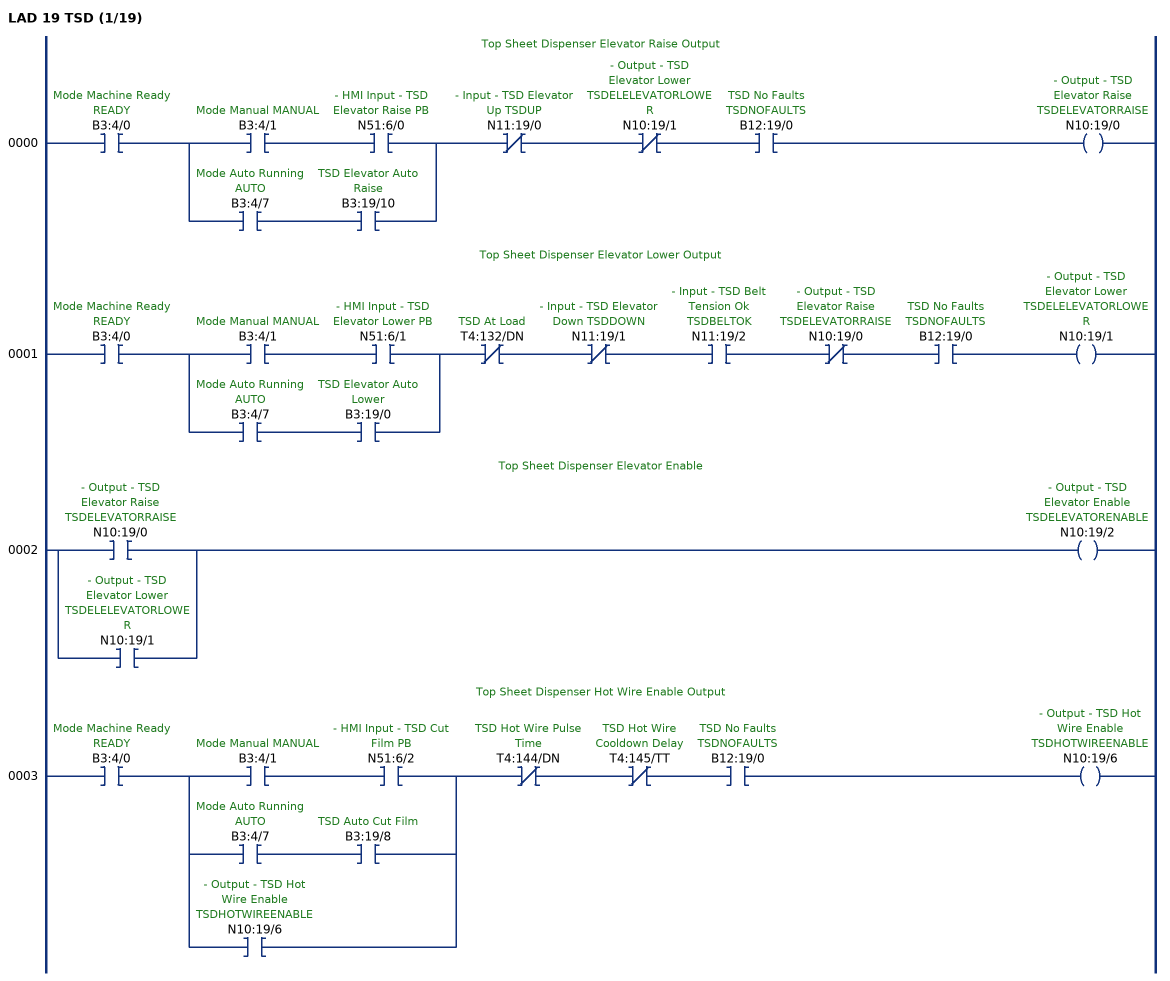
% Rung: 0 %
% Top Sheet Dispenser Elevator Raise Output %
SOR XIC B3:4/0 BST XIC B3:4/1 XIC N51:6/0 NXB XIC B3:4/7 XIC B3:19/10 BND XIO N11:19/0 XIO N10:19/1 XIC B12:19/0 OTE N10:19/0 EOR
%   B3:4/0  READY  "Mode Machine Ready" %
%   B3:4/1  MANUAL  "Mode Manual" %
%   N51:6/0  "- HMI Input - TSD Elevator Raise PB" %
%   B3:4/7  AUTO  "Mode Auto Running" %
%   B3:19/10  "TSD Elevator Auto Raise" %
%   N11:19/0  TSDUP  "- Input - TSD Elevator Up" %
%   N10:19/1  TSDELELEVATORLOWER  "- Output - TSD Elevator Lower" %
%   B12:19/0  TSDNOFAULTS  "TSD No Faults" %
%   N10:19/0  TSDELEVATORRAISE  "- Output - TSD Elevator Raise" %
% Rung: 1 %
% Top Sheet Dispenser Elevator Lower Output %
SOR XIC B3:4/0 BST XIC B3:4/1 XIC N51:6/1 NXB XIC B3:4/7 XIC B3:19/0 BND XIO T4:132/DN XIO N11:19/1 XIC N11:19/2 XIO N10:19/0 XIC B12:19/0 OTE N10:19/1 EOR
%   B3:4/0  READY  "Mode Machine Ready" %
%   B3:4/1  MANUAL  "Mode Manual" %
%   N51:6/1  "- HMI Input - TSD Elevator Lower PB" %
%   B3:4/7  AUTO  "Mode Auto Running" %
%   B3:19/0  "TSD Elevator Auto Lower" %
%   T4:132  "TSD At Load" %
%   N11:19/1  TSDDOWN  "- Input - TSD Elevator Down" %
%   N11:19/2  TSDBELTOK  "- Input - TSD Belt Tension Ok" %
%   N10:19/0  TSDELEVATORRAISE  "- Output - TSD Elevator Raise" %
%   B12:19/0  TSDNOFAULTS  "TSD No Faults" %
%   N10:19/1  TSDELELEVATORLOWER  "- Output - TSD Elevator Lower" %
% Rung: 2 %
% Top Sheet Dispenser Elevator Enable %
SOR BST XIC N10:19/0 NXB XIC N10:19/1 BND OTE N10:19/2 EOR
%   N10:19/0  TSDELEVATORRAISE  "- Output - TSD Elevator Raise" %
%   N10:19/1  TSDELELEVATORLOWER  "- Output - TSD Elevator Lower" %
%   N10:19/2  TSDELEVATORENABLE  "- Output - TSD Elevator Enable" %
% Rung: 3 %
% Top Sheet Dispenser Hot Wire Enable Output %
SOR XIC B3:4/0 BST XIC B3:4/1 XIC N51:6/2 NXB XIC B3:4/7 XIC B3:19/8 NXB XIC N10:19/6 BND XIO T4:144/DN XIO T4:145/TT XIC B12:19/0 OTE N10:19/6 EOR
%   B3:4/0  READY  "Mode Machine Ready" %
%   B3:4/1  MANUAL  "Mode Manual" %
%   N51:6/2  "- HMI Input - TSD Cut Film PB" %
%   B3:4/7  AUTO  "Mode Auto Running" %
%   B3:19/8  "TSD Auto Cut Film" %
%   N10:19/6  TSDHOTWIREENABLE  "- Output - TSD Hot Wire Enable" %
%   T4:144  "TSD Hot Wire Pulse Time" %
%   T4:145  "TSD Hot Wire Cooldown Delay" %
%   B12:19/0  TSDNOFAULTS  "TSD No Faults" %

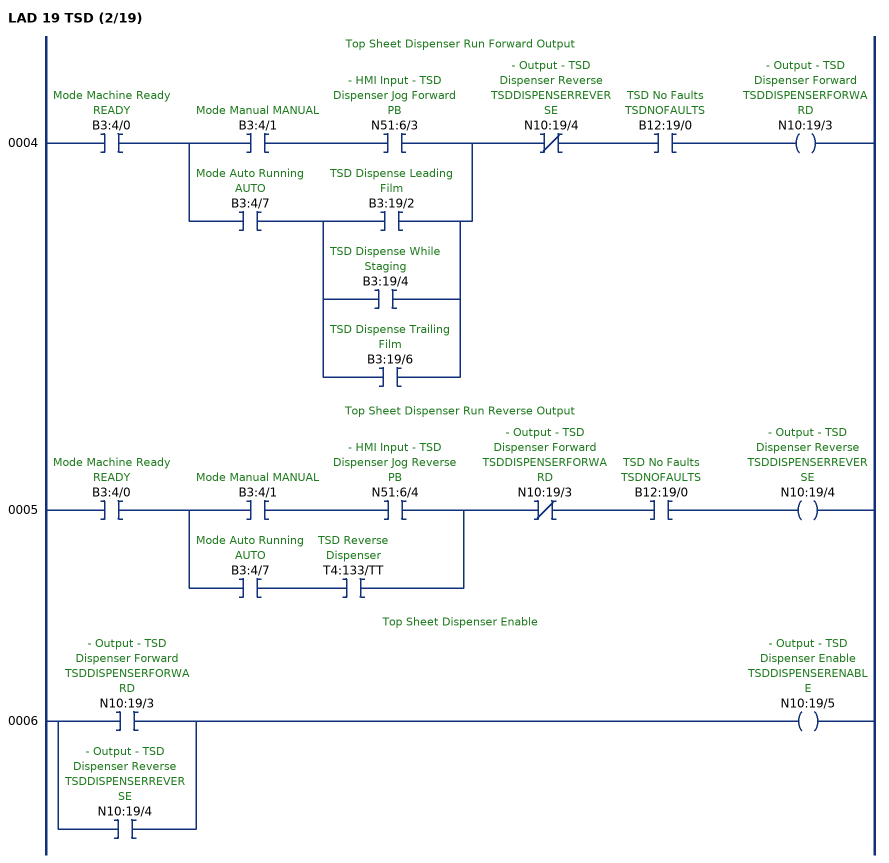
% Rung: 4 %
% Top Sheet Dispenser Run Forward Output %
SOR XIC B3:4/0 BST XIC B3:4/1 XIC N51:6/3 NXB XIC B3:4/7 BST XIC B3:19/2 NXB XIC B3:19/4 NXB XIC B3:19/6 BND BND XIO N10:19/4 XIC B12:19/0 OTE N10:19/3 EOR
%   B3:4/0  READY  "Mode Machine Ready" %
%   B3:4/1  MANUAL  "Mode Manual" %
%   N51:6/3  "- HMI Input - TSD Dispenser Jog Forward PB" %
%   B3:4/7  AUTO  "Mode Auto Running" %
%   B3:19/2  "TSD Dispense Leading Film" %
%   B3:19/4  "TSD Dispense While Staging" %
%   B3:19/6  "TSD Dispense Trailing Film" %
%   N10:19/4  TSDDISPENSERREVERSE  "- Output - TSD Dispenser Reverse" %
%   B12:19/0  TSDNOFAULTS  "TSD No Faults" %
%   N10:19/3  TSDDISPENSERFORWARD  "- Output - TSD Dispenser Forward" %
% Rung: 5 %
% Top Sheet Dispenser Run Reverse Output %
SOR XIC B3:4/0 BST XIC B3:4/1 XIC N51:6/4 NXB XIC B3:4/7 XIC T4:133/TT BND XIO N10:19/3 XIC B12:19/0 OTE N10:19/4 EOR
%   B3:4/0  READY  "Mode Machine Ready" %
%   B3:4/1  MANUAL  "Mode Manual" %
%   N51:6/4  "- HMI Input - TSD Dispenser Jog Reverse PB" %
%   B3:4/7  AUTO  "Mode Auto Running" %
%   T4:133  "TSD Reverse Dispenser" %
%   N10:19/3  TSDDISPENSERFORWARD  "- Output - TSD Dispenser Forward" %
%   B12:19/0  TSDNOFAULTS  "TSD No Faults" %
%   N10:19/4  TSDDISPENSERREVERSE  "- Output - TSD Dispenser Reverse" %
% Rung: 6 %
% Top Sheet Dispenser Enable %
SOR BST XIC N10:19/3 NXB XIC N10:19/4 BND OTE N10:19/5 EOR
%   N10:19/3  TSDDISPENSERFORWARD  "- Output - TSD Dispenser Forward" %
%   N10:19/4  TSDDISPENSERREVERSE  "- Output - TSD Dispenser Reverse" %
%   N10:19/5  TSDDISPENSERENABLE  "- Output - TSD Dispenser Enable" %

